C07193=1038.016,139.466,-96.925,169.847,40.558,157.645
C07194=1038.010,139.217,-96.903,169.845,40.559,157.645
C07195=1038.004,138.968,-96.882,169.843,40.558,157.644
C07196=1037.998,138.720,-96.861,169.840,40.559,157.644
C07197=1037.992,138.470,-96.839,169.837,40.558,157.644
C07198=1037.986,138.221,-96.819,169.835,40.558,157.644
C07199=1037.979,137.972,-96.797,169.833,40.558,157.644
C07200=1037.974,137.723,-96.776,169.831,40.558,157.644
C07201=1037.968,137.474,-96.754,169.828,40.558,157.644
C07202=1037.961,137.225,-96.733,169.826,40.557,157.644
C07203=1037.955,136.976,-96.711,169.824,40.558,157.644
C07204=1037.949,136.727,-96.691,169.822,40.557,157.643
C07205=1037.942,136.478,-96.670,169.819,40.557,157.643
C07206=1037.936,136.229,-96.648,169.817,40.557,157.643
C07207=1037.931,135.980,-96.627,169.814,40.557,157.643
C07208=1037.924,135.731,-96.606,169.812,40.557,157.643
C07209=1037.918,135.481,-96.585,169.810,40.557,157.643
C07210=1037.912,135.233,-96.564,169.807,40.557,157.643
C07211=1037.905,134.984,-96.543,169.805,40.556,157.642
C07212=1037.899,134.735,-96.521,169.803,40.557,157.642
C07213=1037.894,134.486,-96.500,169.801,40.556,157.642
C07214=1037.887,134.237,-96.479,169.799,40.556,157.642
C07215=1037.881,133.987,-96.458,169.796,40.556,157.642
C07216=1037.875,133.739,-96.436,169.793,40.556,157.642
C07217=1037.869,133.489,-96.416,169.791,40.556,157.642
C07218=1037.863,133.240,-96.394,169.789,40.555,157.641
C07219=1037.857,132.992,-96.373,169.787,40.556,157.641
C07220=1037.851,132.742,-96.353,169.784,40.555,157.641
C07221=1037.844,132.493,-96.331,169.782,40.556,157.641
C07222=1037.839,132.245,-96.310,169.780,40.555,157.641
C07223=1037.832,131.995,-96.290,169.778,40.555,157.641
C07224=1037.826,131.746,-96.268,169.776,40.555,157.641
C07225=1037.820,131.498,-96.247,169.773,40.555,157.641
C07226=1037.814,131.248,-96.226,169.770,40.555,157.640
C07227=1037.808,130.999,-96.205,169.768,40.554,157.640
C07228=1037.802,130.750,-96.185,169.766,40.555,157.640
C07229=1037.796,130.501,-96.163,169.764,40.554,157.640
C07230=1037.790,130.252,-96.143,169.762,40.554,157.640
C07231=1037.783,130.003,-96.122,169.759,40.555,157.640
C07232=1037.777,129.753,-96.101,169.757,40.554,157.640
C07233=1037.771,129.505,-96.081,169.755,40.555,157.640
C07234=1037.764,129.255,-96.060,169.753,40.554,157.640
C07235=1037.758,129.006,-96.039,169.750,40.554,157.639
C07236=1037.752,128.757,-96.019,169.748,40.555,157.639
C07237=1037.745,128.508,-95.998,169.745,40.554,157.639
C07238=1037.740,128.259,-95.977,169.743,40.554,157.639
C07239=1037.733,128.010,-95.956,169.741,40.554,157.639
C07240=1037.726,127.761,-95.936,169.738,40.554,157.639
C07241=1037.721,127.512,-95.914,169.736,40.555,157.639
C07242=1037.714,127.263,-95.894,169.734,40.554,157.639
C07243=1037.708,127.015,-95.873,169.732,40.554,157.639
C07244=1037.701,126.765,-95.853,169.730,40.554,157.638
C07245=1037.695,126.515,-95.832,169.728,40.554,157.638
C07246=1037.689,126.267,-95.812,169.725,40.554,157.638
C07247=1037.682,126.018,-95.791,169.722,40.554,157.638
C07248=1037.677,125.769,-95.770,169.720,40.554,157.638
C07249=1037.670,125.520,-95.750,169.718,40.554,157.638
C07250=1037.663,125.234,-95.726,169.715,40.554,157.638
C07251=1037.656,124.949,-95.702,169.713,40.554,157.638
C07252=1037.649,124.662,-95.679,169.710,40.554,157.638
C07253=1037.642,124.377,-95.655,169.708,40.554,157.637
C07254=1037.635,124.127,-95.635,169.706,40.554,157.637
C07255=1037.630,123.879,-95.614,169.704,40.554,157.637
C07256=1037.623,123.629,-95.593,169.701,40.554,157.637
C07257=1037.617,123.380,-95.573,169.699,40.554,157.637
C07258=1037.611,123.131,-95.552,169.696,40.554,157.637
C07259=1037.605,122.882,-95.532,169.694,40.554,157.637
C07260=1037.598,122.633,-95.512,169.692,40.554,157.637
C07261=1037.592,122.385,-95.491,169.690,40.554,157.637
C07262=1037.586,122.135,-95.470,169.687,40.554,157.636
C07263=1037.580,121.886,-95.450,169.685,40.553,157.636
C07264=1037.574,121.636,-95.430,169.683,40.554,157.636
C07265=1037.568,121.388,-95.408,169.681,40.553,157.636
C07266=1037.561,121.138,-95.388,169.679,40.553,157.636
C07267=1037.555,120.890,-95.368,169.677,40.554,157.636
C07268=1037.550,120.641,-95.348,169.675,40.553,157.636
C07269=1037.544,120.391,-95.327,169.672,40.554,157.636
C07270=1037.537,120.143,-95.307,169.669,40.553,157.635
C07271=1037.531,119.893,-95.286,169.667,40.553,157.635
C07272=1037.525,119.644,-95.266,169.665,40.553,157.635
C07273=1037.519,119.395,-95.245,169.663,40.553,157.635
C07274=1037.513,119.146,-95.225,169.661,40.553,157.635
C07275=1037.506,118.897,-95.204,169.659,40.553,157.635
C07276=1037.501,118.648,-95.184,169.657,40.553,157.635
C07277=1037.495,118.399,-95.164,169.654,40.553,157.635
C07278=1037.488,118.149,-95.144,169.652,40.553,157.635
C07279=1037.483,117.900,-95.123,169.650,40.553,157.634
C07280=1037.476,117.651,-95.103,169.648,40.553,157.634
C07281=1037.470,117.403,-95.082,169.645,40.552,157.634
C07282=1037.464,117.154,-95.062,169.643,40.553,157.634
C07283=1037.458,116.904,-95.041,169.641,40.552,157.634
C07284=1037.452,116.655,-95.021,169.639,40.552,157.634
C07285=1037.446,116.406,-95.001,169.637,40.553,157.634
C07286=1037.440,116.157,-94.981,169.634,40.552,157.634
C07287=1037.434,115.908,-94.960,169.632,40.552,157.634
C07288=1037.428,115.658,-94.940,169.630,40.552,157.633
C07289=1037.422,115.409,-94.920,169.628,40.552,157.633
C07290=1037.416,115.161,-94.900,169.626,40.552,157.633
C07291=1037.410,114.911,-94.879,169.624,40.552,157.633
C07292=1037.404,114.662,-94.859,169.621,40.552,157.633
C07293=1037.398,114.413,-94.839,169.619,40.552,157.633
C07294=1037.391,114.164,-94.819,169.617,40.551,157.633
C07295=1037.386,113.915,-94.798,169.615,40.552,157.633
C07296=1037.380,113.666,-94.778,169.612,40.551,157.632
C07297=1037.373,113.417,-94.757,169.610,40.551,157.632
C07298=1037.367,113.167,-94.738,169.608,40.552,157.632
C07299=1037.361,112.919,-94.718,169.606,40.551,157.632
C07300=1037.355,112.669,-94.698,169.604,40.551,157.632
C07301=1037.349,112.420,-94.678,169.602,40.552,157.632
C07302=1037.343,112.171,-94.658,169.600,40.551,157.632
C07303=1037.336,111.922,-94.638,169.598,40.551,157.632
C07304=1037.330,111.673,-94.618,169.595,40.552,157.632
C07305=1037.324,111.424,-94.597,169.592,40.551,157.632
C07306=1037.318,111.175,-94.577,169.590,40.552,157.632
C07307=1037.312,110.925,-94.558,169.588,40.552,157.631
C07308=1037.305,110.676,-94.538,169.586,40.551,157.631
C07309=1037.299,110.427,-94.518,169.584,40.552,157.631
C07310=1037.293,110.178,-94.498,169.582,40.552,157.631
C07311=1037.287,109.929,-94.478,169.580,40.551,157.631
C07312=1037.281,109.680,-94.458,169.578,40.552,157.631
C07313=1037.274,109.431,-94.439,169.575,40.552,157.631
C07314=1037.265,109.034,-94.407,169.572,40.552,157.631
C07315=1037.255,108.637,-94.375,169.569,40.552,157.631
C07316=1037.244,108.240,-94.344,169.565,40.552,157.631
C07317=1037.234,107.844,-94.312,169.561,40.552,157.630
C07318=1037.228,107.595,-94.292,169.559,40.552,157.630
C07319=1037.222,107.346,-94.273,169.557,40.552,157.630
C07320=1037.216,107.097,-94.254,169.555,40.552,157.630
C07321=1037.209,106.847,-94.233,169.553,40.552,157.630
C07322=1037.203,106.599,-94.213,169.550,40.553,157.630
C07323=1037.198,106.349,-94.194,169.548,40.552,157.630
C07324=1037.191,106.100,-94.174,169.546,40.552,157.630
C07325=1037.184,105.851,-94.154,169.544,40.553,157.630
C07326=1037.179,105.602,-94.135,169.542,40.553,157.630
C07327=1037.173,105.353,-94.115,169.540,40.552,157.629
C07328=1037.166,105.103,-94.095,169.538,40.553,157.629
C07329=1037.160,104.854,-94.076,169.536,40.553,157.629
C07330=1037.154,104.605,-94.056,169.533,40.552,157.629
C07331=1037.148,104.357,-94.036,169.531,40.553,157.629
C07332=1037.141,104.106,-94.017,169.528,40.553,157.629
C07333=1037.135,103.858,-93.997,169.526,40.552,157.629
C07334=1037.130,103.608,-93.978,169.524,40.553,157.629
C07335=1037.123,103.360,-93.958,169.522,40.553,157.629
C07336=1037.117,103.111,-93.938,169.520,40.553,157.629
C07337=1037.111,102.861,-93.919,169.518,40.553,157.628
C07338=1037.105,102.612,-93.899,169.516,40.553,157.628
C07339=1037.098,102.363,-93.880,169.514,40.553,157.628
C07340=1037.092,102.114,-93.860,169.512,40.553,157.628
C07341=1037.087,101.865,-93.841,169.510,40.553,157.628
C07342=1037.080,101.615,-93.820,169.508,40.553,157.628
C07343=1037.074,101.366,-93.801,169.506,40.553,157.628
C07344=1037.068,101.117,-93.782,169.503,40.553,157.628
C07345=1037.062,100.868,-93.762,169.500,40.553,157.628
C07346=1037.056,100.619,-93.743,169.498,40.553,157.628
C07347=1037.049,100.369,-93.722,169.496,40.553,157.627
C07348=1037.043,100.120,-93.704,169.494,40.553,157.627
C07349=1037.037,99.871,-93.684,169.492,40.553,157.627
C07350=1037.031,99.622,-93.665,169.490,40.553,157.627
C07351=1037.025,99.373,-93.646,169.488,40.553,157.627
C07352=1037.018,99.123,-93.626,169.486,40.553,157.627
C07353=1037.012,98.874,-93.607,169.484,40.554,157.627
C07354=1037.003,98.487,-93.577,169.480,40.554,157.627
C07355=1036.992,98.100,-93.547,169.477,40.554,157.627
C07356=1036.983,97.712,-93.517,169.474,40.554,157.627
C07357=1036.973,97.324,-93.487,169.471,40.554,157.627
C07358=1036.967,97.075,-93.467,169.468,40.554,157.626
C07359=1036.960,96.826,-93.448,169.466,40.554,157.626
C07360=1036.955,96.576,-93.429,169.463,40.554,157.626
C07361=1036.948,96.328,-93.410,169.461,40.555,157.626
C07362=1036.942,96.078,-93.390,169.459,40.555,157.626
C07363=1036.936,95.829,-93.372,169.457,40.554,157.626
C07364=1036.929,95.579,-93.352,169.455,40.555,157.626
C07365=1036.923,95.331,-93.333,169.453,40.555,157.626
C07366=1036.917,95.081,-93.314,169.451,40.555,157.626
C07367=1036.911,94.832,-93.295,169.449,40.555,157.626
C07368=1036.905,94.583,-93.275,169.447,40.555,157.626
C07369=1036.898,94.334,-93.256,169.445,40.555,157.626
C07370=1036.893,94.085,-93.237,169.442,40.555,157.625
C07371=1036.886,93.836,-93.218,169.440,40.556,157.625
C07372=1036.880,93.587,-93.198,169.438,40.555,157.625
C07373=1036.874,93.338,-93.180,169.436,40.555,157.625
C07374=1036.867,93.051,-93.158,169.434,40.556,157.625
C07375=1036.859,92.766,-93.136,169.431,40.556,157.625
C07376=1036.852,92.479,-93.114,169.429,40.555,157.625
C07377=1036.845,92.194,-93.092,169.426,40.556,157.625
C07378=1036.839,91.944,-93.073,169.424,40.556,157.625
C07379=1036.832,91.695,-93.054,169.422,40.556,157.625
C07380=1036.827,91.446,-93.035,169.419,40.556,157.624
C07381=1036.820,91.197,-93.015,169.417,40.556,157.624
C07382=1036.814,90.948,-92.996,169.415,40.556,157.624
C07383=1036.808,90.699,-92.977,169.413,40.556,157.624
C07384=1036.802,90.449,-92.958,169.411,40.556,157.624
C07385=1036.796,90.200,-92.940,169.409,40.556,157.624
C07386=1036.790,89.951,-92.920,169.407,40.556,157.624
C07387=1036.784,89.702,-92.902,169.405,40.557,157.624
C07388=1036.777,89.452,-92.883,169.403,40.557,157.624
C07389=1036.771,89.203,-92.864,169.401,40.556,157.624
C07390=1036.765,88.954,-92.844,169.399,40.557,157.624
C07391=1036.758,88.705,-92.826,169.397,40.557,157.624
C07392=1036.752,88.456,-92.807,169.395,40.557,157.624
C07393=1036.746,88.207,-92.788,169.392,40.557,157.623
C07394=1036.739,87.958,-92.770,169.390,40.558,157.623
C07395=1036.733,87.708,-92.750,169.388,40.558,157.623
C07396=1036.726,87.459,-92.732,169.386,40.558,157.623
C07397=1036.720,87.210,-92.713,169.384,40.558,157.623
C07398=1036.714,86.960,-92.694,169.381,40.558,157.623
C07399=1036.707,86.711,-92.676,169.379,40.558,157.623
C07400=1036.701,86.462,-92.656,169.377,40.558,157.623
C07401=1036.695,86.213,-92.638,169.375,40.558,157.623
C07402=1036.689,85.963,-92.620,169.373,40.559,157.623
C07403=1036.682,85.714,-92.601,169.371,40.559,157.623
C07404=1036.676,85.465,-92.582,169.368,40.559,157.623
C07405=1036.670,85.215,-92.563,169.366,40.559,157.623
C07406=1036.664,84.966,-92.545,169.364,40.559,157.623
C07407=1036.657,84.717,-92.526,169.362,40.559,157.622
C07408=1036.651,84.468,-92.507,169.360,40.559,157.622
C07409=1036.645,84.219,-92.489,169.358,40.560,157.622
C07410=1036.638,83.970,-92.470,169.356,40.560,157.622
C07411=1036.633,83.720,-92.451,169.354,40.560,157.622
C07412=1036.626,83.471,-92.432,169.352,40.560,157.622
C07413=1036.620,83.221,-92.414,169.350,40.560,157.622
C07414=1036.614,82.973,-92.396,169.348,40.560,157.622
C07415=1036.608,82.724,-92.377,169.346,40.560,157.622
C07416=1036.602,82.475,-92.358,169.344,40.560,157.622
C07417=1036.596,82.225,-92.339,169.341,40.561,157.622
C07418=1036.589,81.976,-92.321,169.338,40.560,157.622
C07419=1036.583,81.727,-92.302,169.336,40.561,157.622
C07420=1036.577,81.477,-92.284,169.334,40.561,157.621
C07421=1036.570,81.228,-92.265,169.332,40.561,157.621
C07422=1036.565,80.979,-92.246,169.330,40.561,157.621
C07423=1036.558,80.730,-92.228,169.328,40.561,157.621
C07424=1036.552,80.481,-92.209,169.326,40.561,157.621
C07425=1036.546,80.231,-92.191,169.324,40.561,157.621
C07426=1036.539,79.982,-92.172,169.322,40.561,157.621
C07427=1036.533,79.733,-92.154,169.320,40.562,157.621
C07428=1036.528,79.484,-92.135,169.318,40.562,157.621
C07429=1036.521,79.235,-92.116,169.316,40.561,157.621
C07430=1036.515,78.985,-92.098,169.314,40.562,157.621
C07431=1036.509,78.736,-92.080,169.312,40.562,157.621
C07432=1036.502,78.487,-92.061,169.310,40.562,157.621
C07433=1036.496,78.237,-92.043,169.307,40.562,157.621
C07434=1036.490,77.988,-92.024,169.305,40.563,157.620
C07435=1036.483,77.739,-92.006,169.303,40.562,157.620
C07436=1036.477,77.490,-91.987,169.301,40.562,157.620
C07437=1036.471,77.241,-91.969,169.299,40.563,157.620
C07438=1036.464,76.954,-91.948,169.297,40.563,157.620
C07439=1036.457,76.669,-91.927,169.293,40.563,157.620
C07440=1036.450,76.383,-91.906,169.291,40.563,157.620
C07441=1036.442,76.096,-91.885,169.289,40.564,157.620
C07442=1036.436,75.848,-91.867,169.287,40.564,157.620
C07443=1036.430,75.599,-91.848,169.284,40.564,157.620
C07444=1036.424,75.349,-91.830,169.282,40.564,157.620
C07445=1036.417,75.100,-91.812,169.280,40.564,157.620
C07446=1036.411,74.850,-91.794,169.278,40.564,157.620
C07447=1036.405,74.601,-91.775,169.276,40.564,157.619
C07448=1036.398,74.351,-91.758,169.274,40.564,157.619
C07449=1036.392,74.103,-91.740,169.272,40.565,157.619
C07450=1036.386,73.854,-91.721,169.270,40.565,157.619
C07451=1036.380,73.604,-91.703,169.268,40.565,157.619
C07452=1036.373,73.355,-91.684,169.266,40.565,157.619
C07453=1036.367,73.105,-91.666,169.264,40.566,157.619
C07454=1036.361,72.856,-91.648,169.262,40.566,157.619
C07455=1036.355,72.607,-91.630,169.259,40.566,157.619
C07456=1036.348,72.358,-91.612,169.257,40.566,157.619
C07457=1036.342,72.108,-91.594,169.255,40.566,157.619
C07458=1036.335,71.859,-91.576,169.253,40.566,157.619
C07459=1036.329,71.610,-91.558,169.251,40.566,157.619
C07460=1036.323,71.361,-91.539,169.249,40.566,157.619
C07461=1036.317,71.111,-91.521,169.247,40.567,157.619
C07462=1036.311,70.862,-91.503,169.245,40.567,157.619
C07463=1036.304,70.613,-91.485,169.243,40.567,157.618
C07464=1036.298,70.363,-91.467,169.241,40.567,157.618
C07465=1036.292,70.115,-91.449,169.239,40.568,157.618
C07466=1036.286,69.865,-91.431,169.237,40.568,157.618
C07467=1036.280,69.616,-91.413,169.234,40.567,157.618
C07468=1036.273,69.366,-91.395,169.231,40.568,157.618
C07469=1036.267,69.117,-91.378,169.229,40.568,157.618
C07470=1036.261,68.868,-91.359,169.227,40.568,157.618
C07471=1036.255,68.619,-91.341,169.225,40.568,157.618
C07472=1036.249,68.369,-91.323,169.223,40.568,157.618
C07473=1036.241,68.120,-91.305,169.221,40.569,157.618
C07474=1036.236,67.871,-91.288,169.219,40.569,157.618
C07475=1036.230,67.621,-91.270,169.217,40.569,157.618
C07476=1036.223,67.372,-91.252,169.215,40.569,157.618
C07477=1036.216,67.123,-91.234,169.213,40.570,157.618
C07478=1036.211,66.874,-91.216,169.211,40.570,157.617
C07479=1036.204,66.625,-91.197,169.209,40.570,157.617
C07480=1036.198,66.375,-91.180,169.206,40.570,157.617
C07481=1036.192,66.125,-91.162,169.204,40.571,157.617
C07482=1036.186,65.877,-91.144,169.202,40.571,157.617
C07483=1036.179,65.627,-91.127,169.200,40.571,157.617
C07484=1036.173,65.378,-91.109,169.198,40.570,157.617
C07485=1036.166,65.129,-91.092,169.196,40.571,157.617
C07486=1036.160,64.880,-91.073,169.194,40.571,157.617
C07487=1036.154,64.630,-91.055,169.192,40.571,157.617
C07488=1036.147,64.381,-91.038,169.190,40.571,157.617
C07489=1036.142,64.132,-91.020,169.188,40.572,157.617
C07490=1036.135,63.882,-91.002,169.186,40.572,157.617
C07491=1036.128,63.633,-90.984,169.183,40.572,157.617
C07492=1036.122,63.383,-90.966,169.181,40.572,157.617
C07493=1036.116,63.135,-90.949,169.179,40.573,157.617
C07494=1036.109,62.885,-90.932,169.177,40.573,157.616
C07495=1036.103,62.635,-90.914,169.175,40.574,157.617
C07496=1036.097,62.387,-90.897,169.173,40.574,157.616
C07497=1036.091,62.137,-90.879,169.171,40.574,157.616
C07498=1036.084,61.888,-90.862,169.169,40.574,157.616
C07499=1036.077,61.638,-90.844,169.166,40.575,157.616
C07500=1036.071,61.389,-90.827,169.164,40.575,157.616
C07501=1036.064,61.140,-90.809,169.162,40.575,157.616
C07502=1036.057,60.854,-90.789,169.160,40.575,157.616
C07503=1036.050,60.568,-90.768,169.156,40.576,157.616
C07504=1036.043,60.282,-90.749,169.154,40.576,157.616
C07505=1036.034,59.995,-90.729,169.151,40.576,157.616
C07506=1036.029,59.746,-90.711,169.150,40.577,157.616
C07507=1036.022,59.497,-90.694,169.148,40.577,157.616
C07508=1036.015,59.248,-90.677,169.146,40.577,157.616
C07509=1036.010,58.999,-90.659,169.143,40.578,157.616
C07510=1036.003,58.749,-90.642,169.141,40.578,157.616
C07511=1035.997,58.499,-90.624,169.139,40.578,157.616
C07512=1035.990,58.251,-90.607,169.136,40.578,157.616
C07513=1035.983,58.001,-90.589,169.134,40.579,157.616
C07514=1035.977,57.751,-90.571,169.132,40.579,157.616
C07515=1035.971,57.503,-90.555,169.130,40.579,157.615
C07516=1035.964,57.253,-90.537,169.128,40.579,157.615
C07517=1035.958,57.003,-90.520,169.126,40.579,157.615
C07518=1035.952,56.754,-90.503,169.124,40.580,157.615
C07519=1035.945,56.505,-90.486,169.122,40.580,157.615
C07520=1035.939,56.255,-90.468,169.120,40.580,157.615
C07521=1035.933,56.006,-90.451,169.117,40.580,157.615
C07522=1035.926,55.757,-90.433,169.115,40.581,157.615
C07523=1035.921,55.508,-90.416,169.113,40.581,157.615
C07524=1035.914,55.258,-90.399,169.111,40.581,157.615
C07525=1035.907,55.009,-90.381,169.109,40.581,157.615
C07526=1035.901,54.760,-90.364,169.107,40.582,157.615
C07527=1035.895,54.510,-90.347,169.105,40.582,157.615
C07528=1035.889,54.261,-90.330,169.103,40.582,157.615
C07529=1035.882,54.011,-90.312,169.100,40.583,157.615
C07530=1035.876,53.763,-90.295,169.098,40.583,157.615
C07531=1035.869,53.513,-90.278,169.096,40.583,157.615
C07532=1035.863,53.264,-90.260,169.094,40.583,157.615
C07533=1035.857,53.015,-90.243,169.092,40.584,157.615
C07534=1035.850,52.765,-90.226,169.090,40.584,157.615
C07535=1035.845,52.516,-90.209,169.088,40.584,157.614
C07536=1035.838,52.266,-90.191,169.086,40.584,157.614
C07537=1035.832,52.018,-90.174,169.084,40.584,157.614
C07538=1035.826,51.768,-90.156,169.081,40.585,157.614
C07539=1035.820,51.518,-90.140,169.079,40.585,157.614
C07540=1035.813,51.269,-90.123,169.077,40.585,157.614
C07541=1035.807,51.020,-90.105,169.075,40.585,157.614
C07542=1035.800,50.771,-90.088,169.073,40.586,157.614
C07543=1035.794,50.521,-90.072,169.071,40.586,157.614
C07544=1035.788,50.272,-90.054,169.069,40.586,157.614
C07545=1035.782,50.023,-90.037,169.067,40.586,157.614
C07546=1035.775,49.773,-90.019,169.065,40.587,157.614
C07547=1035.769,49.524,-90.003,169.063,40.587,157.614
C07548=1035.763,49.274,-89.985,169.060,40.586,157.614
C07549=1035.757,49.025,-89.968,169.058,40.587,157.614
C07550=1035.750,48.776,-89.951,169.055,40.587,157.613
C07551=1035.745,48.526,-89.934,169.053,40.587,157.613
C07552=1035.738,48.277,-89.917,169.051,40.587,157.613
C07553=1035.732,48.028,-89.900,169.049,40.587,157.613
C07554=1035.725,47.778,-89.883,169.047,40.588,157.613
C07555=1035.720,47.529,-89.866,169.045,40.588,157.613
C07556=1035.713,47.280,-89.849,169.043,40.588,157.613
C07557=1035.707,47.030,-89.832,169.040,40.588,157.613
C07558=1035.701,46.781,-89.814,169.038,40.589,157.613
C07559=1035.694,46.532,-89.797,169.036,40.589,157.613
C07560=1035.688,46.283,-89.781,169.034,40.589,157.613
C07561=1035.682,46.033,-89.763,169.032,40.589,157.613
C07562=1035.676,45.784,-89.746,169.030,40.589,157.613
C07563=1035.670,45.535,-89.730,169.028,40.590,157.613
C07564=1035.663,45.285,-89.712,169.026,40.590,157.613
C07565=1035.658,45.036,-89.695,169.024,40.590,157.613
C07566=1035.650,44.749,-89.676,169.021,40.590,157.613
C07567=1035.643,44.463,-89.657,169.019,40.591,157.613
C07568=1035.636,44.177,-89.637,169.016,40.590,157.612
C07569=1035.630,43.890,-89.617,169.014,40.591,157.612
C07570=1035.623,43.640,-89.601,169.012,40.591,157.612
C07571=1035.617,43.391,-89.584,169.010,40.591,157.612
C07572=1035.611,43.142,-89.566,169.008,40.591,157.612
C07573=1035.605,42.892,-89.550,169.006,40.591,157.612
C07574=1035.599,42.643,-89.533,169.003,40.592,157.612
C07575=1035.592,42.394,-89.516,169.001,40.592,157.612
C07576=1035.586,42.144,-89.500,168.999,40.592,157.612
C07577=1035.579,41.895,-89.482,168.997,40.592,157.612
C07578=1035.573,41.645,-89.466,168.995,40.593,157.612
C07579=1035.567,41.397,-89.449,168.993,40.593,157.612
C07580=1035.560,41.147,-89.432,168.991,40.594,157.612
C07581=1035.554,40.898,-89.416,168.988,40.594,157.612
C07582=1035.547,40.648,-89.399,168.986,40.594,157.612
C07583=1035.541,40.399,-89.383,168.984,40.594,157.612
C07584=1035.535,40.150,-89.366,168.982,40.595,157.612
C07585=1035.529,39.900,-89.349,168.980,40.595,157.611
C07586=1035.522,39.651,-89.332,168.978,40.595,157.611
C07587=1035.516,39.402,-89.316,168.976,40.595,157.611
C07588=1035.510,39.152,-89.299,168.973,40.596,157.611
C07589=1035.504,38.903,-89.282,168.970,40.596,157.611
C07590=1035.498,38.654,-89.266,168.968,40.596,157.611
C07591=1035.491,38.404,-89.249,168.966,40.596,157.611
C07592=1035.485,38.155,-89.232,168.964,40.596,157.611
C07593=1035.479,37.905,-89.216,168.962,40.597,157.611
C07594=1035.472,37.655,-89.199,168.960,40.597,157.611
C07595=1035.466,37.407,-89.183,168.957,40.597,157.611
C07596=1035.460,37.157,-89.166,168.955,40.597,157.611
C07597=1035.454,36.907,-89.150,168.953,40.598,157.611
C07598=1035.447,36.658,-89.134,168.951,40.598,157.611
C07599=1035.441,36.410,-89.117,168.949,40.599,157.611
C07600=1035.434,36.159,-89.100,168.947,40.599,157.611
C07601=1035.428,35.910,-89.084,168.944,40.599,157.611
C07602=1035.422,35.661,-89.068,168.942,40.599,157.611
C07603=1035.415,35.411,-89.052,168.940,40.600,157.611
C07604=1035.409,35.162,-89.035,168.938,40.600,157.611
C07605=1035.403,34.913,-89.019,168.936,40.601,157.611
C07606=1035.396,34.663,-89.002,168.934,40.601,157.610
C07607=1035.390,34.414,-88.986,168.931,40.601,157.610
C07608=1035.384,34.165,-88.970,168.929,40.601,157.610
C07609=1035.377,33.915,-88.953,168.927,40.602,157.610
C07610=1035.371,33.666,-88.936,168.925,40.602,157.610
C07611=1035.365,33.416,-88.920,168.923,40.603,157.610
C07612=1035.358,33.167,-88.905,168.920,40.603,157.610
C07613=1035.352,32.917,-88.888,168.918,40.603,157.610
C07614=1035.346,32.668,-88.872,168.916,40.603,157.610
C07615=1035.340,32.419,-88.855,168.914,40.604,157.610
C07616=1035.333,32.170,-88.840,168.912,40.604,157.610
C07617=1035.326,31.920,-88.822,168.910,40.604,157.610
C07618=1035.320,31.671,-88.806,168.907,40.604,157.610
C07619=1035.314,31.421,-88.790,168.905,40.605,157.610
C07620=1035.308,31.172,-88.774,168.903,40.605,157.610
C07621=1035.301,30.922,-88.758,168.901,40.606,157.610
C07622=1035.295,30.673,-88.741,168.899,40.606,157.610
C07623=1035.289,30.424,-88.725,168.896,40.606,157.610
C07624=1035.282,30.175,-88.709,168.894,40.606,157.610
C07625=1035.276,29.925,-88.693,168.892,40.607,157.610
C07626=1035.270,29.675,-88.677,168.890,40.607,157.610
C07627=1035.264,29.426,-88.660,168.888,40.607,157.609
C07628=1035.257,29.177,-88.645,168.886,40.607,157.609
C07629=1035.251,28.927,-88.628,168.883,40.608,157.609
C07630=1035.244,28.641,-88.610,168.881,40.608,157.609
C07631=1035.237,28.354,-88.590,168.878,40.609,157.609
C07632=1035.230,28.067,-88.572,168.876,40.609,157.609
C07633=1035.222,27.781,-88.554,168.873,40.609,157.609
C07634=1035.215,27.532,-88.538,168.871,40.610,157.609
C07635=1035.209,27.282,-88.522,168.869,40.610,157.609
C07636=1035.203,27.033,-88.506,168.867,40.611,157.609
C07637=1035.197,26.784,-88.490,168.865,40.611,157.609
C07638=1035.190,26.534,-88.473,168.862,40.611,157.609
C07639=1035.184,26.284,-88.458,168.860,40.611,157.609
C07640=1035.178,26.035,-88.442,168.858,40.612,157.609
C07641=1035.171,25.786,-88.426,168.856,40.612,157.609
C07642=1035.165,25.537,-88.410,168.853,40.613,157.609
C07643=1035.158,25.287,-88.394,168.851,40.613,157.609
C07644=1035.152,25.038,-88.378,168.849,40.613,157.609
C07645=1035.145,24.789,-88.362,168.847,40.613,157.609
C07646=1035.140,24.539,-88.347,168.845,40.614,157.609
C07647=1035.133,24.290,-88.331,168.842,40.615,157.609
C07648=1035.127,24.040,-88.315,168.840,40.615,157.609
C07649=1035.120,23.791,-88.299,168.838,40.615,157.609
C07650=1035.114,23.541,-88.282,168.836,40.615,157.609
C07651=1035.107,23.292,-88.267,168.833,40.616,157.608
C07652=1035.102,23.042,-88.251,168.831,40.616,157.609
C07653=1035.095,22.793,-88.235,168.829,40.617,157.608
C07654=1035.089,22.544,-88.219,168.827,40.617,157.608
C07655=1035.082,22.295,-88.204,168.825,40.617,157.608
C07656=1035.077,22.045,-88.188,168.822,40.617,157.608
C07657=1035.070,21.796,-88.172,168.820,40.618,157.608
C07658=1035.063,21.546,-88.156,168.818,40.618,157.608
C07659=1035.057,21.297,-88.140,168.816,40.619,157.608
C07660=1035.051,21.047,-88.125,168.813,40.619,157.608
C07661=1035.044,20.798,-88.109,168.811,40.619,157.608
C07662=1035.038,20.548,-88.093,168.809,40.619,157.608
C07663=1035.032,20.299,-88.077,168.807,40.620,157.608
C07664=1035.026,20.049,-88.061,168.805,40.621,157.608
C07665=1035.019,19.800,-88.046,168.802,40.621,157.608
C07666=1035.013,19.551,-88.029,168.800,40.621,157.608
C07667=1035.007,19.301,-88.015,168.798,40.621,157.608
C07668=1035.000,19.052,-87.999,168.796,40.621,157.608
C07669=1034.995,18.802,-87.983,168.793,40.622,157.608
C07670=1034.987,18.552,-87.967,168.791,40.623,157.608
C07671=1034.981,18.303,-87.952,168.789,40.623,157.608
C07672=1034.975,18.053,-87.936,168.787,40.623,157.608
C07673=1034.968,17.804,-87.920,168.784,40.624,157.608
C07674=1034.962,17.555,-87.905,168.782,40.624,157.608
C07675=1034.956,17.305,-87.889,168.780,40.625,157.608
C07676=1034.949,17.056,-87.874,168.778,40.625,157.608
C07677=1034.944,16.806,-87.858,168.775,40.625,157.607
C07678=1034.937,16.557,-87.842,168.773,40.626,157.608
C07679=1034.931,16.308,-87.827,168.771,40.626,157.608
C07680=1034.925,16.058,-87.811,168.769,40.626,157.607
C07681=1034.918,15.809,-87.796,168.766,40.627,157.607
C07682=1034.912,15.560,-87.781,168.764,40.627,157.607
C07683=1034.906,15.310,-87.764,168.762,40.628,157.607
C07684=1034.899,15.061,-87.749,168.760,40.628,157.607
C07685=1034.893,14.812,-87.734,168.757,40.628,157.607
C07686=1034.887,14.562,-87.718,168.755,40.628,157.607
C07687=1034.880,14.313,-87.702,168.753,40.629,157.607
C07688=1034.874,14.063,-87.688,168.751,40.630,157.607
C07689=1034.868,13.813,-87.672,168.748,40.630,157.607
C07690=1034.862,13.564,-87.656,168.746,40.630,157.607
C07691=1034.855,13.314,-87.641,168.744,40.631,157.607
C07692=1034.848,13.065,-87.626,168.741,40.631,157.607
C07693=1034.842,12.816,-87.611,168.739,40.632,157.607
C07694=1034.835,12.530,-87.593,168.737,40.632,157.607
C07695=1034.827,12.245,-87.575,168.734,40.633,157.607
C07696=1034.820,11.959,-87.558,168.731,40.633,157.607
C07697=1034.813,11.675,-87.541,168.729,40.634,157.607
C07698=1034.806,11.425,-87.526,168.726,40.634,157.607
C07699=1034.800,11.176,-87.511,168.725,40.635,157.607
C07700=1034.793,10.926,-87.496,168.723,40.635,157.607
C07701=1034.787,10.677,-87.481,168.719,40.636,157.607
C07702=1034.780,10.428,-87.465,168.718,40.636,157.607
C07703=1034.774,10.178,-87.450,168.716,40.637,157.607
C07704=1034.768,9.928,-87.435,168.713,40.637,157.607
C07705=1034.761,9.679,-87.419,168.711,40.638,157.607
C07706=1034.754,9.430,-87.404,168.709,40.638,157.607
C07707=1034.749,9.180,-87.389,168.707,40.638,157.607
C07708=1034.742,8.930,-87.374,168.704,40.639,157.607
C07709=1034.736,8.681,-87.358,168.702,40.640,157.607
C07710=1034.729,8.431,-87.343,168.700,40.640,157.607
C07711=1034.723,8.182,-87.328,168.697,40.640,157.607
C07712=1034.717,7.932,-87.313,168.695,40.641,157.607
C07713=1034.710,7.683,-87.298,168.693,40.641,157.607
C07714=1034.704,7.433,-87.283,168.690,40.641,157.606
C07715=1034.698,7.184,-87.268,168.688,40.642,157.607
C07716=1034.691,6.935,-87.253,168.686,40.643,157.607
C07717=1034.685,6.686,-87.238,168.683,40.643,157.606
C07718=1034.678,6.436,-87.223,168.681,40.644,157.606
C07719=1034.672,6.186,-87.208,168.679,40.644,157.606
C07720=1034.665,5.937,-87.193,168.676,40.644,157.606
C07721=1034.659,5.687,-87.178,168.674,40.644,157.606
C07722=1034.652,5.438,-87.162,168.672,40.645,157.606
C07723=1034.647,5.189,-87.148,168.670,40.646,157.606
C07724=1034.640,4.939,-87.133,168.667,40.646,157.606
C07725=1034.634,4.690,-87.118,168.665,40.647,157.606
C07726=1034.627,4.440,-87.103,168.663,40.647,157.606
C07727=1034.621,4.191,-87.088,168.660,40.647,157.606
C07728=1034.615,3.941,-87.073,168.658,40.648,157.606
C07729=1034.609,3.692,-87.058,168.656,40.648,157.606
C07730=1034.602,3.443,-87.043,168.653,40.649,157.606
C07731=1034.597,3.193,-87.027,168.651,40.649,157.606
C07732=1034.590,2.943,-87.012,168.649,40.650,157.606
C07733=1034.584,2.694,-86.997,168.646,40.650,157.606
C07734=1034.577,2.444,-86.982,168.644,40.650,157.606
C07735=1034.572,2.195,-86.968,168.642,40.651,157.606
C07736=1034.565,1.945,-86.953,168.639,40.652,157.606
C07737=1034.559,1.696,-86.938,168.637,40.652,157.606
C07738=1034.553,1.446,-86.923,168.635,40.652,157.606
C07739=1034.547,1.197,-86.908,168.632,40.653,157.606
C07740=1034.540,0.947,-86.893,168.630,40.653,157.606
C07741=1034.534,0.698,-86.878,168.628,40.653,157.606
C07742=1034.528,0.448,-86.863,168.625,40.654,157.606
C07743=1034.521,0.198,-86.849,168.623,40.655,157.606
C07744=1034.515,-0.051,-86.834,168.621,40.655,157.606
C07745=1034.509,-0.300,-86.819,168.618,40.655,157.606
C07746=1034.503,-0.550,-86.804,168.616,40.655,157.606
C07747=1034.496,-0.800,-86.789,168.614,40.656,157.606
C07748=1034.491,-1.048,-86.775,168.612,40.656,157.606
C07749=1034.484,-1.298,-86.760,168.609,40.657,157.605
C07750=1034.478,-1.548,-86.745,168.607,40.657,157.605
C07751=1034.472,-1.797,-86.730,168.605,40.658,157.605
C07752=1034.466,-2.046,-86.715,168.602,40.658,157.605
C07753=1034.459,-2.296,-86.700,168.600,40.658,157.605
C07754=1034.453,-2.546,-86.685,168.598,40.659,157.605
C07755=1034.447,-2.795,-86.671,168.595,40.660,157.605
C07756=1034.441,-3.044,-86.656,168.593,40.660,157.605
C07757=1034.434,-3.294,-86.641,168.591,40.660,157.605
C07758=1034.427,-3.577,-86.624,168.588,40.660,157.605
C07759=1034.420,-3.861,-86.608,168.585,40.661,157.605
C07760=1034.413,-4.144,-86.592,168.582,40.662,157.605
C07761=1034.406,-4.427,-86.575,168.580,40.662,157.605
C07762=1034.399,-4.677,-86.561,168.577,40.663,157.605
C07763=1034.393,-4.926,-86.546,168.576,40.664,157.605
C07764=1034.387,-5.176,-86.531,168.574,40.664,157.605
C07765=1034.380,-5.425,-86.517,168.571,40.664,157.605
C07766=1034.374,-5.674,-86.503,168.569,40.665,157.605
C07767=1034.368,-5.924,-86.488,168.566,40.665,157.605
C07768=1034.361,-6.174,-86.474,168.564,40.666,157.605
C07769=1034.354,-6.423,-86.459,168.562,40.666,157.605
C07770=1034.349,-6.673,-86.445,168.559,40.667,157.605
C07771=1034.342,-6.922,-86.431,168.557,40.668,157.605
C07772=1034.335,-7.172,-86.416,168.554,40.668,157.605
C07773=1034.329,-7.421,-86.401,168.552,40.669,157.605
C07774=1034.323,-7.671,-86.388,168.550,40.669,157.605
C07775=1034.316,-7.921,-86.373,168.547,40.670,157.605
C07776=1034.310,-8.170,-86.358,168.545,40.670,157.605
C07777=1034.304,-8.419,-86.344,168.542,40.671,157.605
C07778=1034.297,-8.669,-86.330,168.540,40.671,157.605
C07779=1034.291,-8.918,-86.316,168.538,40.672,157.605
C07780=1034.285,-9.168,-86.301,168.535,40.673,157.605
C07781=1034.279,-9.417,-86.287,168.533,40.673,157.605
C07782=1034.272,-9.667,-86.273,168.530,40.674,157.605
C07783=1034.266,-9.917,-86.258,168.528,40.674,157.605
C07784=1034.260,-10.166,-86.244,168.525,40.674,157.605
C07785=1034.253,-10.416,-86.230,168.523,40.675,157.605
C07786=1034.247,-10.665,-86.215,168.521,40.675,157.605
C07787=1034.241,-10.915,-86.201,168.518,40.676,157.605
C07788=1034.234,-11.164,-86.187,168.516,40.677,157.605
C07789=1034.228,-11.413,-86.172,168.513,40.677,157.605
C07790=1034.221,-11.663,-86.159,168.511,40.678,157.605
C07791=1034.216,-11.912,-86.144,168.509,40.678,157.605
C07792=1034.210,-12.162,-86.130,168.507,40.679,157.605
C07793=1034.202,-12.412,-86.115,168.504,40.679,157.605
C07794=1034.197,-12.661,-86.102,168.501,40.680,157.605
C07795=1034.191,-12.911,-86.087,168.500,40.680,157.605
C07796=1034.184,-13.160,-86.073,168.497,40.681,157.605
C07797=1034.178,-13.410,-86.058,168.495,40.682,157.605
C07798=1034.172,-13.659,-86.045,168.493,40.682,157.605
C07799=1034.165,-13.909,-86.030,168.490,40.682,157.604
C07800=1034.160,-14.158,-86.016,168.488,40.683,157.605
C07801=1034.153,-14.408,-86.002,168.485,40.683,157.604
C07802=1034.147,-14.657,-85.988,168.483,40.684,157.604
C07803=1034.140,-14.907,-85.974,168.481,40.684,157.604
C07804=1034.135,-15.156,-85.960,168.478,40.685,157.604
C07805=1034.128,-15.406,-85.945,168.476,40.686,157.604
C07806=1034.122,-15.655,-85.932,168.473,40.686,157.604
C07807=1034.115,-15.905,-85.918,168.471,40.687,157.604
C07808=1034.109,-16.155,-85.903,168.468,40.687,157.604
C07809=1034.103,-16.404,-85.890,168.466,40.688,157.604
C07810=1034.096,-16.654,-85.876,168.463,40.688,157.604
C07811=1034.090,-16.903,-85.862,168.461,40.689,157.604
C07812=1034.083,-17.153,-85.848,168.458,40.690,157.604
C07813=1034.078,-17.402,-85.834,168.456,40.690,157.604
C07814=1034.071,-17.652,-85.820,168.453,40.691,157.604
C07815=1034.065,-17.901,-85.806,168.451,40.692,157.604
C07816=1034.058,-18.151,-85.792,168.448,40.693,157.604
C07817=1034.052,-18.400,-85.778,168.446,40.693,157.604
C07818=1034.045,-18.650,-85.765,168.444,40.694,157.604
C07819=1034.040,-18.899,-85.751,168.441,40.694,157.604
C07820=1034.033,-19.149,-85.736,168.440,40.695,157.604
C07821=1034.026,-19.398,-85.723,168.437,40.695,157.604
C07822=1034.019,-19.681,-85.708,168.434,40.696,157.604
C07823=1034.012,-19.962,-85.692,168.431,40.697,157.604
C07824=1034.005,-20.243,-85.676,168.429,40.697,157.604
C07825=1033.998,-20.525,-85.661,168.426,40.698,157.604
C07826=1033.992,-20.775,-85.647,168.423,40.699,157.604
C07827=1033.985,-21.024,-85.633,168.421,40.700,157.604
C07828=1033.979,-21.273,-85.619,168.418,40.700,157.604
C07829=1033.973,-21.524,-85.605,168.416,40.701,157.604
C07830=1033.967,-21.773,-85.592,168.413,40.701,157.604
C07831=1033.960,-22.023,-85.578,168.411,40.702,157.604
C07832=1033.955,-22.272,-85.564,168.408,40.702,157.604
C07833=1033.948,-22.521,-85.550,168.406,40.703,157.604
C07834=1033.941,-22.771,-85.537,168.403,40.704,157.604
C07835=1033.935,-23.020,-85.523,168.401,40.704,157.604
C07836=1033.929,-23.271,-85.509,168.398,40.705,157.604
C07837=1033.923,-23.520,-85.496,168.396,40.706,157.604
C07838=1033.917,-23.769,-85.483,168.393,40.706,157.604
C07839=1033.911,-24.019,-85.468,168.391,40.707,157.604
C07840=1033.904,-24.268,-85.455,168.388,40.707,157.604
C07841=1033.898,-24.517,-85.441,168.387,40.708,157.604
C07842=1033.892,-24.768,-85.427,168.384,40.708,157.604
C07843=1033.885,-25.017,-85.414,168.382,40.709,157.604
C07844=1033.879,-25.266,-85.400,168.379,40.710,157.604
C07845=1033.873,-25.516,-85.386,168.377,40.710,157.604
C07846=1033.867,-25.766,-85.373,168.374,40.711,157.604
C07847=1033.861,-26.015,-85.360,168.372,40.712,157.604
C07848=1033.855,-26.265,-85.345,168.369,40.712,157.604
C07849=1033.848,-26.514,-85.332,168.367,40.713,157.604
C07850=1033.842,-26.764,-85.319,168.364,40.713,157.604
C07851=1033.835,-27.014,-85.305,168.362,40.714,157.604
C07852=1033.830,-27.263,-85.291,168.359,40.714,157.604
C07853=1033.824,-27.513,-85.278,168.357,40.715,157.604
C07854=1033.817,-27.763,-85.265,168.354,40.716,157.604
C07855=1033.811,-28.012,-85.251,168.352,40.716,157.604
C07856=1033.804,-28.261,-85.238,168.349,40.717,157.604
C07857=1033.798,-28.511,-85.224,168.347,40.718,157.604
C07858=1033.791,-28.760,-85.211,168.344,40.719,157.604
C07859=1033.785,-29.010,-85.198,168.343,40.720,157.604
C07860=1033.779,-29.260,-85.185,168.340,40.721,157.604
C07861=1033.773,-29.509,-85.172,168.337,40.721,157.604
C07862=1033.766,-29.759,-85.158,168.335,40.722,157.604
C07863=1033.760,-30.009,-85.145,168.332,40.722,157.604
C07864=1033.753,-30.258,-85.131,168.330,40.723,157.604
C07865=1033.747,-30.507,-85.118,168.327,40.724,157.604
C07866=1033.741,-30.756,-85.105,168.325,40.724,157.604
C07867=1033.734,-31.007,-85.092,168.322,40.725,157.604
C07868=1033.728,-31.256,-85.079,168.319,40.726,157.604
C07869=1033.722,-31.505,-85.065,168.317,40.726,157.604
C07870=1033.715,-31.755,-85.052,168.314,40.727,157.604
C07871=1033.709,-32.005,-85.039,168.312,40.728,157.604
C07872=1033.704,-32.255,-85.025,168.309,40.729,157.604
C07873=1033.698,-32.504,-85.012,168.307,40.729,157.604
C07874=1033.691,-32.753,-84.999,168.305,40.730,157.604
C07875=1033.684,-33.003,-84.985,168.301,40.731,157.604
C07876=1033.679,-33.253,-84.973,168.300,40.732,157.604
C07877=1033.672,-33.503,-84.959,168.297,40.732,157.604
C07878=1033.666,-33.752,-84.946,168.295,40.733,157.604
C07879=1033.659,-34.002,-84.932,168.292,40.734,157.604
C07880=1033.653,-34.252,-84.920,168.290,40.734,157.604
C07881=1033.647,-34.501,-84.907,168.287,40.735,157.604
C07882=1033.641,-34.750,-84.893,168.284,40.736,157.604
C07883=1033.635,-34.999,-84.880,168.282,40.736,157.604
C07884=1033.629,-35.249,-84.868,168.279,40.737,157.604
C07885=1033.622,-35.499,-84.854,168.277,40.738,157.604
C07886=1033.615,-35.780,-84.840,168.274,40.738,157.604
C07887=1033.608,-36.061,-84.825,168.271,40.739,157.604
C07888=1033.602,-36.342,-84.810,168.268,40.740,157.604
C07889=1033.594,-36.623,-84.796,168.265,40.741,157.604
C07890=1033.588,-36.873,-84.782,168.262,40.742,157.604
C07891=1033.582,-37.122,-84.769,168.261,40.743,157.604
C07892=1033.576,-37.372,-84.757,168.258,40.743,157.604
C07893=1033.570,-37.621,-84.743,168.256,40.744,157.604
C07894=1033.563,-37.871,-84.730,168.253,40.744,157.604
C07895=1033.557,-38.121,-84.717,168.251,40.745,157.604
C07896=1033.551,-38.370,-84.704,168.248,40.746,157.604
C07897=1033.545,-38.620,-84.691,168.245,40.746,157.604
C07898=1033.539,-38.869,-84.678,168.243,40.747,157.604
C07899=1033.533,-39.119,-84.665,168.240,40.748,157.604
C07900=1033.526,-39.368,-84.653,168.238,40.749,157.604
C07901=1033.520,-39.618,-84.640,168.235,40.749,157.604
C07902=1033.513,-39.868,-84.627,168.232,40.750,157.604
C07903=1033.507,-40.118,-84.614,168.230,40.751,157.604
C07904=1033.500,-40.367,-84.601,168.228,40.752,157.604
C07905=1033.494,-40.617,-84.589,168.224,40.753,157.604
C07906=1033.488,-40.866,-84.576,168.223,40.753,157.604
C07907=1033.482,-41.116,-84.563,168.220,40.754,157.604
C07908=1033.475,-41.365,-84.550,168.217,40.755,157.604
C07909=1033.469,-41.615,-84.538,168.215,40.756,157.605
C07910=1033.463,-41.864,-84.524,168.212,40.757,157.604
C07911=1033.457,-42.114,-84.512,168.209,40.758,157.604
C07912=1033.451,-42.363,-84.500,168.207,40.759,157.605
C07913=1033.444,-42.613,-84.486,168.204,40.760,157.605
C07914=1033.438,-42.863,-84.474,168.202,40.760,157.605
C07915=1033.431,-43.113,-84.462,168.199,40.761,157.605
C07916=1033.425,-43.362,-84.449,168.196,40.762,157.605
C07917=1033.419,-43.612,-84.436,168.195,40.763,157.605
C07918=1033.413,-43.861,-84.423,168.192,40.764,157.605
C07919=1033.406,-44.111,-84.411,168.189,40.764,157.605
C07920=1033.400,-44.361,-84.398,168.187,40.765,157.605
C07921=1033.394,-44.610,-84.385,168.184,40.766,157.605
C07922=1033.388,-44.860,-84.372,168.181,40.767,157.605
C07923=1033.382,-45.109,-84.360,168.179,40.767,157.605
C07924=1033.375,-45.359,-84.347,168.176,40.768,157.605
C07925=1033.369,-45.608,-84.335,168.173,40.769,157.605
C07926=1033.363,-45.858,-84.323,168.171,40.770,157.605
C07927=1033.357,-46.108,-84.310,168.168,40.770,157.605
C07928=1033.351,-46.357,-84.297,168.165,40.771,157.605
C07929=1033.344,-46.607,-84.285,168.164,40.772,157.605
C07930=1033.338,-46.857,-84.272,168.161,40.773,157.605
C07931=1033.332,-47.107,-84.260,168.158,40.774,157.605
C07932=1033.326,-47.356,-84.246,168.156,40.774,157.605
C07933=1033.319,-47.605,-84.235,168.153,40.775,157.605
C07934=1033.313,-47.855,-84.222,168.150,40.776,157.605
C07935=1033.308,-48.104,-84.210,168.148,40.777,157.605
C07936=1033.301,-48.353,-84.197,168.145,40.777,157.605
C07937=1033.295,-48.603,-84.185,168.142,40.778,157.605
C07938=1033.289,-48.853,-84.172,168.140,40.779,157.605
C07939=1033.283,-49.103,-84.160,168.137,40.780,157.605
C07940=1033.277,-49.353,-84.147,168.134,40.781,157.605
C07941=1033.271,-49.602,-84.135,168.132,40.782,157.605
C07942=1033.264,-49.851,-84.122,168.130,40.783,157.605
C07943=1033.258,-50.101,-84.110,168.127,40.784,157.605
C07944=1033.252,-50.351,-84.097,168.125,40.784,157.605
C07945=1033.245,-50.601,-84.085,168.122,40.785,157.605
C07946=1033.240,-50.850,-84.073,168.119,40.786,157.605
C07947=1033.233,-51.100,-84.061,168.117,40.787,157.605
C07948=1033.227,-51.349,-84.049,168.114,40.788,157.605
C07949=1033.221,-51.599,-84.037,168.111,40.789,157.605
C07950=1033.213,-51.880,-84.023,168.108,40.790,157.605
C07951=1033.206,-52.161,-84.009,168.106,40.791,157.605
C07952=1033.199,-52.443,-83.996,168.103,40.792,157.605
C07953=1033.191,-52.725,-83.982,168.100,40.793,157.605
C07954=1033.186,-52.974,-83.970,168.097,40.794,157.606
C07955=1033.179,-53.223,-83.958,168.094,40.795,157.606
C07956=1033.173,-53.473,-83.946,168.091,40.796,157.606
C07957=1033.167,-53.723,-83.933,168.089,40.797,157.606
C07958=1033.160,-53.972,-83.921,168.086,40.798,157.606
C07959=1033.153,-54.222,-83.909,168.084,40.799,157.606
C07960=1033.148,-54.472,-83.897,168.081,40.800,157.606
C07961=1033.141,-54.722,-83.885,168.079,40.801,157.606
C07962=1033.135,-54.971,-83.874,168.076,40.802,157.606
C07963=1033.129,-55.221,-83.861,168.073,40.803,157.606
C07964=1033.123,-55.470,-83.849,168.070,40.804,157.606
C07965=1033.116,-55.720,-83.837,168.068,40.805,157.606
C07966=1033.109,-55.969,-83.825,168.065,40.806,157.606
C07967=1033.103,-56.219,-83.813,168.062,40.807,157.606
C07968=1033.098,-56.469,-83.802,168.060,40.808,157.606
C07969=1033.091,-56.718,-83.790,168.057,40.809,157.606
C07970=1033.085,-56.968,-83.777,168.055,40.810,157.606
C07971=1033.078,-57.218,-83.765,168.052,40.811,157.606
C07972=1033.072,-57.467,-83.754,168.049,40.812,157.606
C07973=1033.066,-57.717,-83.741,168.046,40.813,157.606
C07974=1033.060,-57.967,-83.730,168.044,40.814,157.606
C07975=1033.053,-58.216,-83.718,168.041,40.815,157.606
C07976=1033.047,-58.466,-83.706,168.039,40.816,157.606
C07977=1033.041,-58.716,-83.694,168.036,40.817,157.606
C07978=1033.035,-58.965,-83.683,168.034,40.818,157.607
C07979=1033.029,-59.215,-83.671,168.031,40.819,157.607
C07980=1033.022,-59.464,-83.659,168.028,40.820,157.607
C07981=1033.016,-59.714,-83.646,168.025,40.821,157.607
C07982=1033.010,-59.964,-83.635,168.022,40.822,157.607
C07983=1033.004,-60.213,-83.623,168.020,40.822,157.607
C07984=1032.998,-60.463,-83.611,168.017,40.823,157.607
C07985=1032.992,-60.712,-83.599,168.015,40.824,157.607
C07986=1032.985,-60.962,-83.588,168.012,40.825,157.607
C07987=1032.979,-61.212,-83.576,168.010,40.826,157.607
C07988=1032.973,-61.462,-83.564,168.007,40.827,157.607
C07989=1032.967,-61.711,-83.553,168.004,40.828,157.607
C07990=1032.960,-61.961,-83.541,168.001,40.829,157.607
C07991=1032.954,-62.210,-83.529,167.999,40.830,157.607
C07992=1032.949,-62.460,-83.517,167.996,40.831,157.607
C07993=1032.942,-62.710,-83.505,167.993,40.832,157.607
C07994=1032.935,-62.959,-83.493,167.991,40.833,157.607
C07995=1032.930,-63.209,-83.482,167.988,40.834,157.607
C07996=1032.924,-63.459,-83.470,167.986,40.835,157.607
C07997=1032.917,-63.709,-83.459,167.983,40.836,157.607
C07998=1032.911,-63.958,-83.447,167.980,40.837,157.607
C07999=1032.905,-64.207,-83.435,167.977,40.838,157.607
C08000=1032.899,-64.458,-83.423,167.974,40.839,157.607
C08001=1032.893,-64.707,-83.412,167.972,40.840,157.607
C08002=1032.887,-64.957,-83.400,167.970,40.841,157.607
C08003=1032.880,-65.207,-83.388,167.967,40.842,157.608
C08004=1032.874,-65.456,-83.378,167.964,40.843,157.608
C08005=1032.868,-65.706,-83.365,167.962,40.844,157.608
C08006=1032.862,-65.955,-83.353,167.959,40.845,157.608
C08007=1032.856,-66.205,-83.342,167.956,40.846,157.608
C08008=1032.849,-66.455,-83.330,167.953,40.847,157.608
C08009=1032.844,-66.704,-83.319,167.950,40.848,157.608
C08010=1032.838,-66.954,-83.307,167.948,40.849,157.608
C08011=1032.832,-67.203,-83.296,167.946,40.850,157.608
C08012=1032.825,-67.453,-83.284,167.943,40.851,157.608
C08013=1032.820,-67.702,-83.273,167.940,40.852,157.608
C08014=1032.813,-67.985,-83.260,167.937,40.853,157.608
C08015=1032.806,-68.269,-83.247,167.934,40.854,157.608
C08016=1032.799,-68.551,-83.234,167.931,40.855,157.608
C08017=1032.792,-68.834,-83.221,167.928,40.856,157.608
C08018=1032.786,-69.083,-83.209,167.925,40.857,157.608
C08019=1032.780,-69.333,-83.197,167.923,40.858,157.608
C08020=1032.774,-69.582,-83.186,167.920,40.859,157.608
C08021=1032.768,-69.832,-83.175,167.917,40.860,157.608
C08022=1032.762,-70.082,-83.164,167.915,40.861,157.608
C08023=1032.756,-70.331,-83.152,167.912,40.862,157.608
C08024=1032.751,-70.581,-83.140,167.909,40.863,157.608
C08025=1032.744,-70.831,-83.128,167.906,40.864,157.608
C08026=1032.738,-71.080,-83.117,167.903,40.865,157.608
C08027=1032.732,-71.330,-83.106,167.902,40.866,157.609
C08028=1032.726,-71.579,-83.095,167.899,40.867,157.609
C08029=1032.720,-71.829,-83.083,167.896,40.868,157.609
C08030=1032.715,-72.079,-83.072,167.893,40.869,157.609
C08031=1032.708,-72.329,-83.060,167.890,40.870,157.609
C08032=1032.702,-72.578,-83.049,167.888,40.871,157.609
C08033=1032.696,-72.828,-83.038,167.885,40.872,157.609
C08034=1032.690,-73.078,-83.027,167.882,40.873,157.609
C08035=1032.685,-73.327,-83.015,167.879,40.874,157.609
C08036=1032.678,-73.577,-83.003,167.877,40.875,157.609
C08037=1032.673,-73.827,-82.993,167.874,40.876,157.609
C08038=1032.666,-74.076,-82.981,167.872,40.877,157.609
C08039=1032.660,-74.326,-82.970,167.869,40.879,157.609
C08040=1032.655,-74.575,-82.959,167.866,40.880,157.609
C08041=1032.648,-74.826,-82.948,167.863,40.881,157.609
C08042=1032.643,-75.075,-82.937,167.860,40.882,157.609
C08043=1032.636,-75.325,-82.925,167.857,40.883,157.609
C08044=1032.630,-75.574,-82.914,167.855,40.884,157.609
///RCONF 1,0,0,1,0,0,0,0,0,0,0,0,0,0,0,0,0,0,0,0,0,0,0,0
C08045=1032.623,-75.824,-82.903,167.853,40.885,157.609
C08046=1032.617,-76.074,-82.892,167.850,40.886,157.609
C08047=1032.612,-76.323,-82.881,167.847,40.887,157.609
C08048=1032.605,-76.573,-82.870,167.844,40.889,157.610
C08049=1032.599,-76.823,-82.859,167.841,40.890,157.610
C08050=1032.593,-77.073,-82.848,167.839,40.891,157.610
C08051=1032.587,-77.322,-82.837,167.836,40.892,157.610
C08052=1032.582,-77.572,-82.826,167.834,40.893,157.610
C08053=1032.575,-77.822,-82.815,167.831,40.895,157.610
C08054=1032.569,-78.071,-82.805,167.828,40.896,157.610
C08055=1032.563,-78.321,-82.794,167.825,40.897,157.610
C08056=1032.556,-78.570,-82.782,167.822,40.898,157.610
C08057=1032.551,-78.820,-82.771,167.820,40.899,157.610
C08058=1032.544,-79.070,-82.760,167.817,40.900,157.610
C08059=1032.539,-79.319,-82.749,167.814,40.901,157.610
C08060=1032.533,-79.569,-82.738,167.811,40.902,157.610
C08061=1032.527,-79.819,-82.727,167.809,40.903,157.610
C08062=1032.520,-80.068,-82.717,167.806,40.905,157.610
C08063=1032.515,-80.318,-82.706,167.804,40.906,157.611
C08064=1032.508,-80.569,-82.695,167.801,40.907,157.611
C08065=1032.502,-80.818,-82.685,167.798,40.909,157.611
C08066=1032.496,-81.067,-82.674,167.795,40.910,157.611
C08067=1032.489,-81.317,-82.663,167.792,40.911,157.611
C08068=1032.483,-81.567,-82.652,167.789,40.912,157.611
C08069=1032.478,-81.816,-82.642,167.787,40.913,157.611
C08070=1032.470,-82.066,-82.631,167.784,40.915,157.611
C08071=1032.465,-82.316,-82.621,167.781,40.916,157.611
C08072=1032.459,-82.566,-82.610,167.778,40.918,157.611
C08073=1032.452,-82.816,-82.599,167.775,40.919,157.611
///RCONF 1,0,0,0,0,0,0,0,0,0,0,0,0,0,0,0,0,0,0,0,0,0,0,0
C08074=1032.446,-83.065,-82.588,167.773,40.920,157.611
C08075=1032.440,-83.314,-82.578,167.771,40.921,157.612
C08076=1032.434,-83.564,-82.567,167.768,40.922,157.612
C08077=1032.428,-83.815,-82.557,167.765,40.924,157.612
C08078=1032.421,-84.099,-82.544,167.761,40.925,157.612
C08079=1032.414,-84.384,-82.532,167.758,40.927,157.612
C08080=1032.406,-84.668,-82.520,167.756,40.928,157.612
C08081=1032.400,-84.953,-82.508,167.752,40.929,157.612
C08082=1032.394,-85.202,-82.498,167.749,40.931,157.612
C08083=1032.388,-85.453,-82.487,167.746,40.932,157.612
C08084=1032.381,-85.702,-82.477,167.743,40.933,157.612
C08085=1032.376,-85.952,-82.466,167.742,40.935,157.612
C08086=1032.369,-86.202,-82.456,167.739,40.936,157.612
C08087=1032.364,-86.451,-82.445,167.736,40.937,157.612
C08088=1032.357,-86.701,-82.434,167.733,40.938,157.613
C08089=1032.351,-86.950,-82.424,167.730,40.939,157.613
C08090=1032.346,-87.201,-82.414,167.727,40.941,157.613
C08091=1032.339,-87.450,-82.404,167.724,40.942,157.613
C08092=1032.333,-87.700,-82.392,167.722,40.944,157.613
C08093=1032.327,-87.950,-82.383,167.719,40.945,157.613
C08094=1032.321,-88.199,-82.372,167.716,40.946,157.613
C08095=1032.315,-88.449,-82.361,167.713,40.948,157.613
C08096=1032.309,-88.699,-82.351,167.710,40.949,157.613
C08097=1032.303,-88.948,-82.340,167.708,40.950,157.613
C08098=1032.296,-89.199,-82.331,167.705,40.951,157.613
C08099=1032.291,-89.448,-82.320,167.702,40.952,157.613
C08100=1032.284,-89.697,-82.309,167.699,40.954,157.614
C08101=1032.279,-89.947,-82.299,167.696,40.955,157.614
C08102=1032.273,-90.197,-82.288,167.693,40.957,157.614
C08103=1032.267,-90.447,-82.279,167.691,40.958,157.614
C08104=1032.261,-90.696,-82.268,167.689,40.959,157.614
C08105=1032.255,-90.945,-82.258,167.686,40.960,157.614
C08106=1032.249,-91.196,-82.247,167.683,40.961,157.614
C08107=1032.242,-91.445,-82.237,167.680,40.963,157.614
C08108=1032.237,-91.695,-82.227,167.677,40.964,157.614
C08109=1032.231,-91.945,-82.216,167.675,40.966,157.614
C08110=1032.225,-92.195,-82.206,167.672,40.967,157.614
C08111=1032.219,-92.444,-82.195,167.669,40.968,157.615
C08112=1032.213,-92.694,-82.186,167.666,40.969,157.615
C08113=1032.207,-92.943,-82.175,167.663,40.970,157.615
C08114=1032.201,-93.193,-82.165,167.661,40.972,157.615
C08115=1032.195,-93.443,-82.154,167.658,40.973,157.615
C08116=1032.189,-93.693,-82.145,167.655,40.975,157.615
C08117=1032.183,-93.942,-82.134,167.652,40.976,157.615
C08118=1032.177,-94.192,-82.124,167.649,40.977,157.615
C08119=1032.172,-94.442,-82.114,167.646,40.978,157.615
C08120=1032.165,-94.692,-82.104,167.644,40.979,157.615
C08121=1032.159,-94.942,-82.093,167.641,40.981,157.615
C08122=1032.153,-95.191,-82.083,167.638,40.982,157.615
C08123=1032.147,-95.441,-82.073,167.635,40.984,157.615
C08124=1032.142,-95.691,-82.063,167.632,40.985,157.615
C08125=1032.135,-95.940,-82.053,167.630,40.987,157.616
C08126=1032.130,-96.191,-82.042,167.628,40.987,157.616
C08127=1032.123,-96.440,-82.032,167.625,40.989,157.616
C08128=1032.118,-96.690,-82.022,167.622,40.990,157.616
C08129=1032.112,-96.939,-82.013,167.619,40.991,157.616
C08130=1032.107,-97.188,-82.002,167.616,40.993,157.616
C08131=1032.100,-97.438,-81.992,167.614,40.994,157.616
C08132=1032.095,-97.688,-81.982,167.611,40.996,157.616
C08133=1032.089,-97.938,-81.973,167.608,40.997,157.616
C08134=1032.082,-98.187,-81.962,167.605,40.998,157.616
C08135=1032.076,-98.437,-81.953,167.603,41.000,157.617
C08136=1032.071,-98.687,-81.943,167.600,41.001,157.617
C08137=1032.065,-98.937,-81.933,167.597,41.003,157.617
C08138=1032.058,-99.186,-81.923,167.594,41.004,157.617
C08139=1032.052,-99.436,-81.913,167.591,41.005,157.617
C08140=1032.047,-99.686,-81.903,167.589,41.007,157.617
C08141=1032.040,-99.936,-81.893,167.586,41.009,157.617
C08142=1032.034,-100.203,-81.883,167.582,41.010,157.617
C08143=1032.027,-100.469,-81.873,167.579,41.012,157.617
C08144=1032.021,-100.736,-81.861,167.576,41.013,157.617
C08145=1032.015,-101.002,-81.851,167.574,41.015,157.618
C08146=1032.009,-101.252,-81.841,167.571,41.016,157.618
C08147=1032.002,-101.502,-81.832,167.568,41.018,157.618
C08148=1031.997,-101.752,-81.822,167.565,41.019,157.618
C08149=1031.991,-102.002,-81.812,167.562,41.020,157.618
C08150=1031.984,-102.272,-81.802,167.559,41.022,157.618
C08151=1031.977,-102.542,-81.791,167.556,41.024,157.618
C08152=1031.971,-102.812,-81.781,167.553,41.025,157.618
C08153=1031.965,-103.082,-81.769,167.550,41.027,157.618
C08154=1031.959,-103.331,-81.760,167.548,41.028,157.619
C08155=1031.953,-103.581,-81.751,167.544,41.030,157.619
C08156=1031.947,-103.831,-81.741,167.541,41.031,157.619
C08157=1031.941,-104.081,-81.731,167.538,41.033,157.619
C08158=1031.935,-104.330,-81.721,167.536,41.035,157.619
C08159=1031.929,-104.580,-81.712,167.533,41.036,157.619
C08160=1031.923,-104.830,-81.702,167.530,41.037,157.619
C08161=1031.917,-105.079,-81.693,167.527,41.039,157.619
C08162=1031.912,-105.329,-81.683,167.524,41.040,157.619
C08163=1031.906,-105.579,-81.673,167.522,41.042,157.620
C08164=1031.899,-105.829,-81.664,167.519,41.043,157.620
C08165=1031.893,-106.079,-81.654,167.516,41.044,157.620
C08166=1031.888,-106.328,-81.645,167.513,41.046,157.620
C08167=1031.881,-106.578,-81.635,167.510,41.048,157.620
C08168=1031.876,-106.828,-81.625,167.508,41.049,157.620
C08169=1031.870,-107.078,-81.616,167.505,41.051,157.620
C08170=1031.864,-107.328,-81.607,167.502,41.052,157.620
C08171=1031.858,-107.577,-81.598,167.499,41.054,157.620
C08172=1031.852,-107.827,-81.588,167.496,41.055,157.620
C08173=1031.846,-108.077,-81.579,167.494,41.057,157.621
C08174=1031.840,-108.326,-81.569,167.491,41.058,157.621
C08175=1031.834,-108.576,-81.559,167.488,41.060,157.621
C08176=1031.828,-108.825,-81.550,167.486,41.062,157.621
C08177=1031.822,-109.076,-81.541,167.483,41.063,157.621
C08178=1031.816,-109.325,-81.532,167.480,41.064,157.621
C08179=1031.810,-109.575,-81.522,167.476,41.066,157.621
C08180=1031.804,-109.824,-81.513,167.473,41.068,157.621
C08181=1031.798,-110.074,-81.503,167.471,41.070,157.622
C08182=1031.792,-110.325,-81.495,167.468,41.071,157.622
C08183=1031.786,-110.574,-81.485,167.465,41.072,157.622
C08184=1031.781,-110.823,-81.476,167.462,41.074,157.622
C08185=1031.774,-111.073,-81.466,167.460,41.076,157.622
C08186=1031.769,-111.324,-81.457,167.457,41.077,157.622
C08187=1031.762,-111.574,-81.448,167.454,41.079,157.622
C08188=1031.757,-111.823,-81.439,167.451,41.080,157.622
C08189=1031.751,-112.072,-81.429,167.449,41.082,157.623
C08190=1031.745,-112.323,-81.420,167.446,41.084,157.623
C08191=1031.739,-112.572,-81.411,167.443,41.085,157.623
C08192=1031.733,-112.822,-81.401,167.440,41.087,157.623
C08193=1031.727,-113.072,-81.393,167.437,41.088,157.623
C08194=1031.722,-113.321,-81.383,167.434,41.090,157.623
C08195=1031.715,-113.571,-81.374,167.431,41.092,157.623
C08196=1031.709,-113.821,-81.364,167.428,41.093,157.623
C08197=1031.704,-114.071,-81.356,167.426,41.095,157.624
C08198=1031.698,-114.320,-81.346,167.423,41.097,157.624
C08199=1031.692,-114.571,-81.337,167.420,41.098,157.624
C08200=1031.686,-114.820,-81.328,167.417,41.099,157.624
C08201=1031.680,-115.070,-81.319,167.414,41.101,157.624
C08202=1031.674,-115.320,-81.310,167.412,41.103,157.624
C08203=1031.669,-115.569,-81.301,167.409,41.105,157.624
C08204=1031.663,-115.820,-81.292,167.406,41.106,157.624
C08205=1031.657,-116.068,-81.283,167.403,41.108,157.625
C08206=1031.650,-116.355,-81.272,167.400,41.110,157.625
C08207=1031.643,-116.642,-81.262,167.396,41.112,157.625
C08208=1031.636,-116.928,-81.252,167.393,41.113,157.625
C08209=1031.630,-117.214,-81.241,167.390,41.116,157.625
C08210=1031.624,-117.465,-81.232,167.387,41.117,157.625
C08211=1031.618,-117.714,-81.224,167.384,41.119,157.625
C08212=1031.612,-117.964,-81.215,167.381,41.120,157.626
C08213=1031.606,-118.214,-81.205,167.379,41.122,157.626
C08214=1031.600,-118.464,-81.197,167.376,41.124,157.626
C08215=1031.594,-118.713,-81.187,167.373,41.125,157.626
C08216=1031.589,-118.963,-81.179,167.370,41.127,157.626
C08217=1031.582,-119.213,-81.170,167.368,41.129,157.626
C08218=1031.577,-119.462,-81.161,167.364,41.131,157.626
C08219=1031.571,-119.712,-81.152,167.361,41.132,157.626
C08220=1031.565,-119.962,-81.143,167.358,41.134,157.627
C08221=1031.560,-120.212,-81.135,167.356,41.136,157.627
C08222=1031.553,-120.462,-81.126,167.353,41.137,157.627
C08223=1031.547,-120.711,-81.117,167.350,41.139,157.627
C08224=1031.541,-120.961,-81.107,167.348,41.141,157.627
C08225=1031.536,-121.211,-81.099,167.345,41.143,157.627
C08226=1031.529,-121.461,-81.091,167.342,41.144,157.627
C08227=1031.524,-121.710,-81.082,167.339,41.146,157.628
C08228=1031.518,-121.961,-81.073,167.336,41.148,157.628
C08229=1031.513,-122.210,-81.064,167.333,41.149,157.628
C08230=1031.506,-122.460,-81.055,167.330,41.151,157.628
C08231=1031.500,-122.709,-81.047,167.327,41.153,157.628
C08232=1031.495,-122.960,-81.038,167.325,41.155,157.628
C08233=1031.489,-123.209,-81.029,167.322,41.156,157.628
C08234=1031.482,-123.459,-81.020,167.319,41.158,157.629
C08235=1031.477,-123.709,-81.012,167.316,41.160,157.629
C08236=1031.472,-123.958,-81.003,167.314,41.161,157.629
C08237=1031.466,-124.208,-80.994,167.310,41.163,157.629
C08238=1031.460,-124.458,-80.986,167.307,41.165,157.629
C08239=1031.454,-124.708,-80.977,167.305,41.167,157.629
C08240=1031.449,-124.958,-80.969,167.302,41.168,157.629
C08241=1031.442,-125.207,-80.960,167.299,41.171,157.630
C08242=1031.436,-125.457,-80.951,167.296,41.173,157.630
C08243=1031.430,-125.707,-80.943,167.294,41.174,157.630
C08244=1031.425,-125.957,-80.934,167.291,41.176,157.630
C08245=1031.419,-126.207,-80.926,167.287,41.178,157.630
C08246=1031.413,-126.457,-80.918,167.285,41.179,157.630
C08247=1031.407,-126.706,-80.909,167.282,41.181,157.631
C08248=1031.400,-126.956,-80.900,167.279,41.183,157.631
C08249=1031.395,-127.206,-80.892,167.276,41.185,157.631
C08250=1031.390,-127.455,-80.883,167.274,41.187,157.631
C08251=1031.384,-127.705,-80.875,167.271,41.189,157.631
C08252=1031.378,-127.954,-80.866,167.267,41.191,157.631
C08253=1031.373,-128.204,-80.857,167.265,41.191,157.631
C08254=1031.368,-128.454,-80.847,167.263,41.193,157.631
C08255=1031.365,-128.703,-80.837,167.259,41.193,157.631
C08256=1031.362,-128.953,-80.826,167.257,41.192,157.631
C08257=1031.360,-129.203,-80.815,167.255,41.192,157.631
C08258=1031.357,-129.453,-80.803,167.253,41.191,157.631
C08259=1031.356,-129.703,-80.790,167.250,41.190,157.630
C08260=1031.355,-129.952,-80.777,167.249,41.187,157.630
C08261=1031.355,-130.202,-80.763,167.246,41.185,157.629
C08262=1031.357,-130.453,-80.748,167.244,41.182,157.629
C08263=1031.357,-130.702,-80.734,167.243,41.179,157.628
C08264=1031.360,-130.953,-80.718,167.242,41.175,157.627
C08265=1031.362,-131.202,-80.702,167.240,41.171,157.626
C08266=1031.366,-131.452,-80.685,167.239,41.166,157.626
C08267=1031.370,-131.703,-80.668,167.237,41.160,157.625
C08268=1031.374,-131.952,-80.650,167.236,41.155,157.624
C08269=1031.380,-132.202,-80.631,167.235,41.149,157.623
C08270=1031.057,-132.227,-80.929,167.185,41.384,157.659
C08271=1031.051,-131.977,-80.947,167.187,41.390,157.660
C08272=1031.047,-131.727,-80.966,167.188,41.396,157.661
C08273=1031.043,-131.477,-80.983,167.189,41.401,157.662
C08274=1031.040,-131.227,-80.999,167.190,41.406,157.663
C08275=1031.037,-130.977,-81.016,167.192,41.410,157.664
C08276=1031.035,-130.727,-81.031,167.194,41.414,157.665
C08277=1031.033,-130.477,-81.046,167.196,41.417,157.665
C08278=1031.033,-130.227,-81.060,167.198,41.421,157.666
C08279=1031.033,-129.978,-81.075,167.200,41.423,157.666
C08280=1031.033,-129.728,-81.088,167.202,41.425,157.667
C08281=1031.034,-129.478,-81.101,167.204,41.426,157.667
C08282=1031.037,-129.228,-81.113,167.206,41.428,157.668
C08283=1031.039,-128.978,-81.124,167.208,41.428,157.668
C08284=1031.042,-128.728,-81.135,167.211,41.428,157.668
C08285=1031.046,-128.479,-81.145,167.213,41.428,157.668
C08286=1031.050,-128.230,-81.156,167.216,41.427,157.668
C08287=1031.054,-127.980,-81.165,167.219,41.426,157.668
C08288=1031.060,-127.730,-81.173,167.222,41.424,157.668
C08289=1031.066,-127.480,-81.181,167.225,41.423,157.668
C08290=1031.073,-127.231,-81.190,167.227,41.420,157.668
C08291=1031.078,-126.981,-81.199,167.230,41.418,157.667
C08292=1031.084,-126.731,-81.207,167.234,41.417,157.667
C08293=1031.090,-126.481,-81.215,167.236,41.415,157.667
C08294=1031.095,-126.232,-81.224,167.239,41.413,157.667
C08295=1031.102,-125.982,-81.232,167.242,41.411,157.667
C08296=1031.107,-125.732,-81.241,167.244,41.409,157.667
C08297=1031.113,-125.482,-81.250,167.247,41.407,157.667
C08298=1031.119,-125.233,-81.258,167.250,41.405,157.666
C08299=1031.125,-124.982,-81.267,167.254,41.404,157.666
C08300=1031.131,-124.733,-81.275,167.256,41.402,157.666
C08301=1031.136,-124.484,-81.284,167.259,41.400,157.666
C08302=1031.142,-124.233,-81.293,167.262,41.398,157.666
C08303=1031.148,-123.984,-81.301,167.265,41.397,157.666
C08304=1031.154,-123.733,-81.310,167.267,41.394,157.665
C08305=1031.160,-123.484,-81.319,167.271,41.392,157.665
C08306=1031.166,-123.234,-81.328,167.274,41.391,157.665
C08307=1031.172,-122.985,-81.335,167.276,41.389,157.665
C08308=1031.177,-122.734,-81.344,167.279,41.387,157.665
C08309=1031.183,-122.485,-81.354,167.282,41.386,157.665
C08310=1031.188,-122.235,-81.362,167.284,41.384,157.665
C08311=1031.195,-121.985,-81.370,167.287,41.382,157.665
C08312=1031.200,-121.736,-81.379,167.290,41.380,157.664
C08313=1031.206,-121.486,-81.388,167.294,41.378,157.664
C08314=1031.212,-121.236,-81.397,167.296,41.377,157.664
C08315=1031.218,-120.987,-81.406,167.299,41.375,157.664
C08316=1031.224,-120.737,-81.414,167.302,41.373,157.664
C08317=1031.230,-120.486,-81.423,167.305,41.372,157.664
C08318=1031.235,-120.237,-81.432,167.307,41.370,157.664
C08319=1031.241,-119.987,-81.441,167.310,41.368,157.663
C08320=1031.248,-119.737,-81.450,167.313,41.366,157.663
C08321=1031.253,-119.488,-81.459,167.316,41.365,157.663
C08322=1031.259,-119.237,-81.467,167.319,41.363,157.663
C08323=1031.265,-118.988,-81.477,167.322,41.361,157.663
C08324=1031.271,-118.738,-81.485,167.325,41.359,157.663
C08325=1031.277,-118.489,-81.494,167.327,41.358,157.663
C08326=1031.283,-118.239,-81.503,167.330,41.356,157.663
C08327=1031.288,-117.989,-81.512,167.333,41.354,157.662
C08328=1031.294,-117.739,-81.521,167.336,41.352,157.662
C08329=1031.300,-117.489,-81.531,167.339,41.351,157.662
C08330=1031.306,-117.240,-81.539,167.342,41.349,157.662
C08331=1031.313,-116.953,-81.549,167.345,41.347,157.662
C08332=1031.319,-116.667,-81.560,167.348,41.345,157.662
C08333=1031.326,-116.380,-81.569,167.351,41.343,157.661
C08334=1031.333,-116.094,-81.580,167.355,41.341,157.661
C08335=1031.339,-115.845,-81.590,167.357,41.339,157.661
C08336=1031.344,-115.594,-81.598,167.360,41.338,157.661
C08337=1031.351,-115.345,-81.607,167.363,41.336,157.661
C08338=1031.357,-115.095,-81.616,167.366,41.334,157.661
C08339=1031.363,-114.845,-81.625,167.369,41.332,157.661
C08340=1031.369,-114.595,-81.634,167.372,41.331,157.661
C08341=1031.374,-114.346,-81.643,167.375,41.329,157.660
C08342=1031.380,-114.096,-81.653,167.378,41.327,157.660
C08343=1031.386,-113.846,-81.662,167.380,41.325,157.660
C08344=1031.392,-113.596,-81.671,167.383,41.324,157.660
C08345=1031.398,-113.347,-81.681,167.386,41.323,157.660
C08346=1031.404,-113.096,-81.689,167.389,41.321,157.660
C08347=1031.409,-112.847,-81.699,167.391,41.319,157.660
C08348=1031.416,-112.597,-81.708,167.394,41.318,157.660
C08349=1031.421,-112.347,-81.717,167.398,41.316,157.659
C08350=1031.427,-112.098,-81.726,167.401,41.314,157.659
C08351=1031.433,-111.848,-81.736,167.403,41.312,157.659
C08352=1031.439,-111.598,-81.745,167.406,41.311,157.659
C08353=1031.445,-111.349,-81.754,167.409,41.309,157.659
C08354=1031.451,-111.099,-81.763,167.412,41.308,157.659
C08355=1031.457,-110.849,-81.773,167.414,41.306,157.659
C08356=1031.462,-110.599,-81.782,167.417,41.304,157.659
C08357=1031.468,-110.349,-81.791,167.420,41.303,157.658
C08358=1031.475,-110.100,-81.801,167.422,41.301,157.658
C08359=1031.481,-109.850,-81.810,167.425,41.299,157.658
C08360=1031.486,-109.601,-81.819,167.429,41.298,157.658
C08361=1031.492,-109.350,-81.828,167.432,41.296,157.658
C08362=1031.498,-109.100,-81.838,167.435,41.295,157.658
C08363=1031.505,-108.851,-81.847,167.437,41.293,157.658
C08364=1031.510,-108.602,-81.857,167.440,41.291,157.658
C08365=1031.516,-108.352,-81.866,167.443,41.289,157.657
C08366=1031.522,-108.101,-81.875,167.445,41.288,157.657
C08367=1031.528,-107.852,-81.885,167.448,41.287,157.657
C08368=1031.534,-107.602,-81.894,167.451,41.285,157.657
C08369=1031.540,-107.353,-81.903,167.454,41.283,157.657
C08370=1031.546,-107.103,-81.913,167.457,41.282,157.657
C08371=1031.552,-106.853,-81.923,167.459,41.280,157.657
C08372=1031.558,-106.603,-81.933,167.463,41.279,157.657
C08373=1031.563,-106.354,-81.942,167.466,41.277,157.657
C08374=1031.570,-106.104,-81.951,167.469,41.275,157.656
C08375=1031.576,-105.854,-81.961,167.471,41.273,157.656
C08376=1031.582,-105.604,-81.971,167.474,41.272,157.656
C08377=1031.588,-105.354,-81.979,167.477,41.271,157.656
C08378=1031.593,-105.105,-81.989,167.480,41.269,157.656
C08379=1031.599,-104.855,-81.999,167.482,41.267,157.656
C08380=1031.605,-104.605,-82.008,167.485,41.266,157.656
C08381=1031.611,-104.355,-82.018,167.488,41.265,157.656
C08382=1031.617,-104.105,-82.027,167.491,41.263,157.656
C08383=1031.623,-103.855,-82.038,167.494,41.262,157.656
C08384=1031.629,-103.607,-82.048,167.496,41.260,157.655
C08385=1031.635,-103.357,-82.057,167.499,41.258,157.655
C08386=1031.641,-103.107,-82.067,167.502,41.257,157.655
C08387=1031.647,-102.858,-82.076,167.505,41.256,157.655
C08388=1031.653,-102.607,-82.086,167.507,41.254,157.655
C08389=1031.659,-102.358,-82.096,167.510,41.252,157.655
C08390=1031.665,-102.108,-82.106,167.513,41.251,157.655
C08391=1031.671,-101.858,-82.115,167.517,41.249,157.655
C08392=1031.676,-101.609,-82.125,167.519,41.248,157.654
C08393=1031.682,-101.359,-82.134,167.522,41.247,157.654
C08394=1031.688,-101.109,-82.144,167.525,41.245,157.654
C08395=1031.696,-100.822,-82.155,167.528,41.243,157.654
C08396=1031.702,-100.535,-82.167,167.532,41.241,157.654
C08397=1031.709,-100.248,-82.179,167.534,41.240,157.654
C08398=1031.716,-99.961,-82.190,167.538,41.238,157.654
C08399=1031.722,-99.712,-82.199,167.541,41.236,157.654
C08400=1031.728,-99.462,-82.209,167.544,41.235,157.654
C08401=1031.734,-99.212,-82.219,167.546,41.233,157.653
C08402=1031.740,-98.963,-82.229,167.549,41.232,157.653
C08403=1031.746,-98.713,-82.239,167.552,41.231,157.653
C08404=1031.752,-98.463,-82.249,167.555,41.229,157.653
C08405=1031.758,-98.213,-82.258,167.557,41.227,157.653
C08406=1031.764,-97.963,-82.268,167.560,41.226,157.653
C08407=1031.771,-97.714,-82.278,167.563,41.224,157.653
C08408=1031.776,-97.464,-82.288,167.566,41.223,157.653
C08409=1031.782,-97.214,-82.298,167.569,41.222,157.653
C08410=1031.788,-96.964,-82.309,167.571,41.220,157.653
C08411=1031.794,-96.715,-82.318,167.574,41.219,157.653
C08412=1031.799,-96.465,-82.329,167.577,41.217,157.652
C08413=1031.806,-96.215,-82.339,167.580,41.216,157.652
C08414=1031.811,-95.965,-82.349,167.583,41.215,157.652
C08415=1031.818,-95.715,-82.359,167.586,41.213,157.652
C08416=1031.823,-95.466,-82.370,167.588,41.212,157.652
C08417=1031.829,-95.216,-82.379,167.591,41.211,157.652
C08418=1031.835,-94.966,-82.389,167.594,41.209,157.652
C08419=1031.841,-94.717,-82.400,167.597,41.208,157.652
C08420=1031.847,-94.467,-82.410,167.599,41.206,157.652
C08421=1031.853,-94.218,-82.420,167.602,41.205,157.652
C08422=1031.859,-93.968,-82.430,167.605,41.204,157.652
C08423=1031.864,-93.718,-82.441,167.608,41.203,157.652
C08424=1031.871,-93.468,-82.451,167.611,41.201,157.651
C08425=1031.876,-93.218,-82.461,167.614,41.200,157.651
C08426=1031.883,-92.969,-82.471,167.616,41.198,157.651
C08427=1031.888,-92.719,-82.481,167.619,41.197,157.651
C08428=1031.894,-92.470,-82.491,167.622,41.195,157.651
C08429=1031.900,-92.220,-82.502,167.625,41.194,157.651
C08430=1031.906,-91.970,-82.512,167.628,41.193,157.651
C08431=1031.912,-91.720,-82.522,167.630,41.192,157.651
C08432=1031.918,-91.471,-82.532,167.633,41.191,157.651
C08433=1031.924,-91.220,-82.543,167.636,41.189,157.651
C08434=1031.931,-90.971,-82.553,167.639,41.188,157.651
C08435=1031.937,-90.722,-82.564,167.642,41.186,157.651
C08436=1031.942,-90.471,-82.574,167.645,41.185,157.650
C08437=1031.948,-90.222,-82.585,167.647,41.183,157.650
C08438=1031.954,-89.972,-82.595,167.649,41.182,157.650
C08439=1031.960,-89.723,-82.605,167.652,41.181,157.650
C08440=1031.966,-89.473,-82.615,167.655,41.180,157.650
C08441=1031.973,-89.223,-82.626,167.657,41.178,157.650
C08442=1031.979,-88.974,-82.637,167.660,41.177,157.650
C08443=1031.984,-88.723,-82.647,167.663,41.175,157.650
C08444=1031.991,-88.474,-82.657,167.666,41.174,157.650
C08445=1031.996,-88.224,-82.667,167.669,41.173,157.650
C08446=1032.002,-87.975,-82.678,167.672,41.172,157.650
C08447=1032.009,-87.725,-82.689,167.674,41.170,157.649
C08448=1032.015,-87.475,-82.698,167.677,41.169,157.649
C08449=1032.021,-87.225,-82.709,167.680,41.167,157.649
C08450=1032.026,-86.976,-82.720,167.683,41.166,157.649
C08451=1032.036,-86.630,-82.734,167.687,41.164,157.649
C08452=1032.043,-86.284,-82.748,167.690,41.162,157.649
C08453=1032.052,-85.938,-82.763,167.695,41.161,157.649
C08454=1032.061,-85.592,-82.778,167.699,41.159,157.649
C08455=1032.066,-85.373,-82.787,167.700,41.157,157.649
C08456=1032.071,-85.154,-82.797,167.703,41.156,157.649
C08457=1032.077,-84.935,-82.805,167.705,41.155,157.649
C08458=1032.082,-84.715,-82.815,167.708,41.154,157.649
C08459=1032.087,-84.497,-82.824,167.711,41.152,157.648
C08460=1032.092,-84.277,-82.834,167.713,41.152,157.648
C08461=1032.098,-84.059,-82.842,167.716,41.151,157.648
C08462=1032.103,-83.839,-82.852,167.717,41.149,157.648
C08463=1032.109,-83.590,-82.863,167.720,41.148,157.648
C08464=1032.115,-83.340,-82.873,167.723,41.147,157.648
C08465=1032.122,-83.090,-82.884,167.726,41.145,157.648
C08466=1032.128,-82.841,-82.894,167.729,41.144,157.648
C08467=1032.134,-82.591,-82.905,167.731,41.142,157.648
C08468=1032.140,-82.341,-82.916,167.734,41.141,157.648
C08469=1032.146,-82.091,-82.926,167.737,41.140,157.648
C08470=1032.152,-81.842,-82.937,167.740,41.139,157.648
C08471=1032.158,-81.592,-82.948,167.743,41.137,157.647
C08472=1032.165,-81.342,-82.958,167.746,41.136,157.647
C08473=1032.171,-81.093,-82.969,167.748,41.134,157.647
C08474=1032.178,-80.843,-82.980,167.751,41.133,157.647
C08475=1032.183,-80.594,-82.991,167.754,41.132,157.647
C08476=1032.189,-80.344,-83.001,167.757,41.131,157.647
C08477=1032.196,-80.094,-83.011,167.760,41.130,157.647
C08478=1032.202,-79.844,-83.022,167.762,41.128,157.647
C08479=1032.207,-79.595,-83.033,167.765,41.127,157.647
C08480=1032.214,-79.344,-83.044,167.768,41.126,157.647
C08481=1032.220,-79.095,-83.055,167.771,41.124,157.647
C08482=1032.225,-78.845,-83.066,167.773,41.123,157.647
C08483=1032.232,-78.596,-83.077,167.776,41.122,157.647
C08484=1032.238,-78.346,-83.088,167.778,41.120,157.646
C08485=1032.244,-78.097,-83.099,167.781,41.119,157.646
C08486=1032.250,-77.846,-83.110,167.784,41.118,157.646
C08487=1032.256,-77.597,-83.121,167.787,41.117,157.646
C08488=1032.262,-77.348,-83.132,167.790,41.116,157.646
C08489=1032.268,-77.098,-83.144,167.793,41.115,157.646
C08490=1032.274,-76.848,-83.154,167.796,41.114,157.646
C08491=1032.281,-76.598,-83.165,167.798,41.113,157.646
C08492=1032.287,-76.349,-83.176,167.800,41.111,157.646
C08493=1032.293,-76.099,-83.187,167.803,41.110,157.646
C08494=1032.299,-75.849,-83.198,167.806,41.109,157.646
C08495=1032.305,-75.600,-83.209,167.809,41.107,157.646
C08496=1032.311,-75.350,-83.220,167.812,41.106,157.646
///RCONF 1,0,0,1,0,0,0,0,0,0,0,0,0,0,0,0,0,0,0,0,0,0,0,0
C08497=1032.317,-75.100,-83.231,167.814,41.105,157.646
C08498=1032.323,-74.851,-83.243,167.817,41.104,157.646
C08499=1032.329,-74.601,-83.254,167.820,41.103,157.645
C08500=1032.335,-74.352,-83.265,167.823,41.102,157.645
C08501=1032.342,-74.102,-83.275,167.825,41.101,157.645
C08502=1032.347,-73.852,-83.287,167.828,41.100,157.645
C08503=1032.354,-73.602,-83.299,167.831,41.099,157.645
C08504=1032.359,-73.353,-83.310,167.833,41.098,157.645
C08505=1032.366,-73.103,-83.321,167.836,41.096,157.645
C08506=1032.371,-72.853,-83.332,167.839,41.095,157.645
C08507=1032.377,-72.604,-83.343,167.841,41.094,157.645
C08508=1032.383,-72.354,-83.355,167.844,41.093,157.645
C08509=1032.389,-72.104,-83.366,167.847,41.092,157.645
C08510=1032.395,-71.855,-83.378,167.850,41.091,157.645
C08511=1032.401,-71.605,-83.389,167.852,41.090,157.645
C08512=1032.408,-71.355,-83.400,167.855,41.089,157.645
C08513=1032.413,-71.106,-83.412,167.857,41.088,157.645
C08514=1032.419,-70.856,-83.424,167.860,41.087,157.645
C08515=1032.425,-70.606,-83.435,167.863,41.086,157.645
C08516=1032.432,-70.357,-83.446,167.866,41.085,157.645
C08517=1032.437,-70.107,-83.457,167.869,41.084,157.645
C08518=1032.444,-69.857,-83.469,167.871,41.082,157.645
C08519=1032.449,-69.608,-83.481,167.873,41.081,157.645
C08520=1032.455,-69.358,-83.492,167.876,41.080,157.645
C08521=1032.461,-69.109,-83.504,167.879,41.079,157.645
C08522=1032.468,-68.858,-83.515,167.882,41.078,157.644
C08523=1032.474,-68.576,-83.528,167.885,41.077,157.644
C08524=1032.481,-68.293,-83.541,167.888,41.076,157.644
C08525=1032.488,-68.010,-83.554,167.890,41.074,157.644
C08526=1032.495,-67.728,-83.567,167.894,41.073,157.644
C08527=1032.501,-67.479,-83.578,167.896,41.072,157.644
C08528=1032.507,-67.229,-83.590,167.899,41.071,157.644
C08529=1032.512,-66.980,-83.602,167.902,41.070,157.644
C08530=1032.519,-66.729,-83.613,167.905,41.069,157.644
C08531=1032.525,-66.480,-83.625,167.908,41.068,157.644
C08532=1032.531,-66.230,-83.636,167.911,41.067,157.644
///RCONF 1,0,0,0,0,0,0,0,0,0,0,0,0,0,0,0,0,0,0,0,0,0,0,0
C08533=1032.538,-65.981,-83.648,167.913,41.066,157.644
C08534=1032.543,-65.731,-83.659,167.915,41.065,157.644
C08535=1032.549,-65.481,-83.671,167.918,41.064,157.644
C08536=1032.556,-65.231,-83.683,167.921,41.063,157.644
C08537=1032.562,-64.982,-83.694,167.924,41.062,157.644
C08538=1032.567,-64.732,-83.706,167.926,41.061,157.644
C08539=1032.573,-64.483,-83.718,167.929,41.060,157.644
C08540=1032.580,-64.233,-83.730,167.932,41.059,157.644
C08541=1032.586,-63.983,-83.741,167.934,41.058,157.644
C08542=1032.592,-63.734,-83.753,167.937,41.057,157.644
C08543=1032.598,-63.484,-83.764,167.939,41.056,157.644
C08544=1032.605,-63.234,-83.776,167.942,41.055,157.644
C08545=1032.611,-62.985,-83.788,167.945,41.054,157.643
C08546=1032.617,-62.735,-83.799,167.948,41.053,157.643
C08547=1032.623,-62.485,-83.812,167.951,41.052,157.643
C08548=1032.629,-62.236,-83.822,167.954,41.051,157.643
C08549=1032.635,-61.986,-83.834,167.955,41.049,157.643
C08550=1032.642,-61.737,-83.846,167.958,41.048,157.643
C08551=1032.647,-61.487,-83.858,167.961,41.047,157.643
C08552=1032.654,-61.237,-83.870,167.964,41.046,157.643
C08553=1032.660,-60.988,-83.882,167.967,41.045,157.643
C08554=1032.665,-60.738,-83.893,167.969,41.044,157.643
C08555=1032.672,-60.488,-83.905,167.972,41.043,157.643
C08556=1032.679,-60.239,-83.917,167.975,41.042,157.643
C08557=1032.685,-59.989,-83.929,167.977,41.041,157.643
C08558=1032.690,-59.739,-83.941,167.980,41.040,157.643
C08559=1032.697,-59.490,-83.953,167.982,41.039,157.643
C08560=1032.704,-59.240,-83.965,167.985,41.038,157.643
C08561=1032.710,-58.991,-83.977,167.988,41.037,157.643
C08562=1032.715,-58.741,-83.988,167.991,41.036,157.643
C08563=1032.722,-58.491,-84.000,167.994,41.035,157.643
C08564=1032.728,-58.242,-84.012,167.995,41.034,157.643
C08565=1032.735,-57.992,-84.024,167.998,41.033,157.643
C08566=1032.740,-57.742,-84.035,168.001,41.032,157.643
C08567=1032.747,-57.493,-84.047,168.004,41.031,157.642
C08568=1032.753,-57.243,-84.059,168.006,41.030,157.642
C08569=1032.759,-56.993,-84.072,168.009,41.029,157.642
C08570=1032.766,-56.744,-84.084,168.012,41.028,157.642
C08571=1032.772,-56.494,-84.095,168.015,41.027,157.642
C08572=1032.778,-56.245,-84.107,168.018,41.026,157.642
C08573=1032.784,-55.995,-84.119,168.019,41.025,157.642
C08574=1032.791,-55.745,-84.131,168.022,41.023,157.642
C08575=1032.798,-55.496,-84.143,168.025,41.022,157.642
C08576=1032.803,-55.246,-84.155,168.028,41.021,157.642
C08577=1032.810,-54.997,-84.167,168.031,41.020,157.642
C08578=1032.816,-54.747,-84.178,168.033,41.019,157.642
C08579=1032.822,-54.497,-84.191,168.036,41.018,157.642
C08580=1032.828,-54.247,-84.203,168.038,41.017,157.642
C08581=1032.835,-53.998,-84.215,168.041,41.016,157.642
C08582=1032.842,-53.748,-84.227,168.044,41.015,157.642
C08583=1032.847,-53.499,-84.239,168.046,41.014,157.642
C08584=1032.854,-53.249,-84.251,168.049,41.013,157.642
C08585=1032.860,-53.000,-84.263,168.052,41.012,157.642
C08586=1032.866,-52.750,-84.276,168.055,41.010,157.642
C08587=1032.874,-52.468,-84.289,168.057,41.009,157.641
C08588=1032.881,-52.187,-84.303,168.060,41.008,157.641
C08589=1032.888,-51.905,-84.316,168.063,41.007,157.641
C08590=1032.895,-51.624,-84.329,168.066,41.006,157.641
C08591=1032.901,-51.374,-84.342,168.069,41.005,157.641
C08592=1032.908,-51.125,-84.354,168.072,41.004,157.641
C08593=1032.915,-50.876,-84.366,168.075,41.003,157.641
C08594=1032.920,-50.626,-84.379,168.076,41.002,157.641
C08595=1032.927,-50.376,-84.391,168.079,41.001,157.641
C08596=1032.933,-50.127,-84.403,168.082,41.000,157.641
C08597=1032.939,-49.877,-84.416,168.084,41.000,157.641
C08598=1032.946,-49.627,-84.428,168.087,40.999,157.641
C08599=1032.951,-49.377,-84.441,168.090,40.998,157.641
C08600=1032.957,-49.127,-84.453,168.092,40.997,157.641
C08601=1032.963,-48.879,-84.465,168.095,40.996,157.641
C08602=1032.970,-48.629,-84.478,168.098,40.995,157.641
C08603=1032.976,-48.379,-84.490,168.101,40.994,157.641
C08604=1032.981,-48.129,-84.503,168.103,40.993,157.641
C08605=1032.988,-47.880,-84.515,168.105,40.992,157.641
C08606=1032.994,-47.630,-84.528,168.108,40.991,157.641
C08607=1033.000,-47.381,-84.541,168.110,40.990,157.641
C08608=1033.007,-47.131,-84.553,168.113,40.989,157.641
C08609=1033.013,-46.881,-84.565,168.116,40.989,157.641
C08610=1033.019,-46.631,-84.578,168.118,40.988,157.641
C08611=1033.026,-46.382,-84.591,168.121,40.987,157.641
C08612=1033.032,-46.133,-84.603,168.124,40.986,157.641
C08613=1033.037,-45.883,-84.616,168.126,40.985,157.641
C08614=1033.044,-45.633,-84.628,168.129,40.984,157.641
C08615=1033.050,-45.384,-84.641,168.132,40.984,157.641
C08616=1033.056,-45.134,-84.653,168.133,40.983,157.641
C08617=1033.062,-44.884,-84.666,168.136,40.982,157.641
C08618=1033.069,-44.635,-84.679,168.139,40.981,157.641
C08619=1033.075,-44.385,-84.691,168.142,40.980,157.641
C08620=1033.081,-44.135,-84.704,168.144,40.979,157.641
C08621=1033.088,-43.886,-84.716,168.147,40.978,157.641
C08622=1033.094,-43.637,-84.729,168.150,40.978,157.641
C08623=1033.100,-43.387,-84.742,168.152,40.977,157.641
C08624=1033.106,-43.137,-84.755,168.155,40.976,157.641
C08625=1033.113,-42.888,-84.767,168.158,40.975,157.640
C08626=1033.118,-42.638,-84.779,168.159,40.974,157.640
C08627=1033.125,-42.389,-84.793,168.162,40.973,157.640
C08628=1033.131,-42.139,-84.805,168.165,40.973,157.640
C08629=1033.137,-41.890,-84.818,168.167,40.972,157.640
C08630=1033.143,-41.640,-84.830,168.170,40.971,157.640
C08631=1033.149,-41.390,-84.843,168.173,40.970,157.640
C08632=1033.156,-41.141,-84.856,168.175,40.969,157.640
C08633=1033.163,-40.891,-84.869,168.178,40.968,157.640
C08634=1033.169,-40.641,-84.882,168.181,40.967,157.640
C08635=1033.175,-40.391,-84.894,168.183,40.967,157.640
C08636=1033.182,-40.142,-84.907,168.186,40.966,157.640
C08637=1033.188,-39.893,-84.920,168.188,40.965,157.640
C08638=1033.194,-39.643,-84.932,168.190,40.964,157.640
C08639=1033.200,-39.393,-84.945,168.193,40.963,157.640
C08640=1033.207,-39.144,-84.957,168.196,40.962,157.640
C08641=1033.213,-38.895,-84.971,168.198,40.961,157.640
C08642=1033.220,-38.645,-84.984,168.201,40.960,157.640
C08643=1033.225,-38.395,-84.997,168.204,40.959,157.640
C08644=1033.232,-38.145,-85.010,168.206,40.959,157.640
C08645=1033.238,-37.896,-85.023,168.209,40.958,157.640
C08646=1033.244,-37.646,-85.036,168.211,40.957,157.640
C08647=1033.250,-37.396,-85.048,168.214,40.956,157.640
C08648=1033.256,-37.147,-85.062,168.216,40.955,157.640
C08649=1033.262,-36.898,-85.075,168.218,40.955,157.640
C08650=1033.268,-36.648,-85.088,168.221,40.954,157.640
C08651=1033.276,-36.367,-85.103,168.224,40.953,157.640
C08652=1033.282,-36.086,-85.117,168.227,40.952,157.640
C08653=1033.289,-35.805,-85.133,168.230,40.952,157.640
C08654=1033.296,-35.525,-85.147,168.233,40.951,157.640
C08655=1033.303,-35.275,-85.160,168.235,40.950,157.640
C08656=1033.309,-35.025,-85.173,168.238,40.949,157.640
C08657=1033.315,-34.776,-85.186,168.240,40.949,157.640
C08658=1033.321,-34.526,-85.199,168.243,40.948,157.640
C08659=1033.328,-34.277,-85.213,168.246,40.947,157.640
C08660=1033.333,-34.027,-85.225,168.248,40.946,157.640
C08661=1033.340,-33.777,-85.239,168.250,40.945,157.640
C08662=1033.346,-33.528,-85.252,168.252,40.944,157.640
C08663=1033.352,-33.278,-85.265,168.255,40.943,157.640
C08664=1033.359,-33.029,-85.278,168.258,40.943,157.640
C08665=1033.365,-32.779,-85.292,168.260,40.942,157.640
C08666=1033.372,-32.530,-85.305,168.263,40.941,157.640
C08667=1033.378,-32.280,-85.317,168.265,40.941,157.640
C08668=1033.384,-32.030,-85.331,168.268,40.940,157.640
C08669=1033.390,-31.781,-85.344,168.271,40.939,157.640
C08670=1033.397,-31.531,-85.358,168.273,40.938,157.640
C08671=1033.403,-31.282,-85.371,168.276,40.938,157.640
C08672=1033.409,-31.032,-85.383,168.278,40.937,157.640
C08673=1033.415,-30.783,-85.397,168.280,40.936,157.640
C08674=1033.421,-30.532,-85.411,168.284,40.935,157.640
C08675=1033.427,-30.283,-85.424,168.285,40.935,157.640
C08676=1033.434,-30.034,-85.437,168.288,40.934,157.640
C08677=1033.440,-29.784,-85.451,168.290,40.933,157.640
C08678=1033.446,-29.534,-85.464,168.293,40.932,157.640
C08679=1033.453,-29.285,-85.477,168.295,40.931,157.640
C08680=1033.459,-29.036,-85.490,168.298,40.930,157.640
C08681=1033.466,-28.786,-85.504,168.301,40.929,157.640
C08682=1033.472,-28.536,-85.517,168.303,40.929,157.640
C08683=1033.478,-28.287,-85.530,168.306,40.928,157.640
C08684=1033.485,-28.037,-85.544,168.308,40.927,157.640
C08685=1033.491,-27.788,-85.557,168.311,40.927,157.640
C08686=1033.497,-27.539,-85.570,168.314,40.926,157.640
C08687=1033.504,-27.289,-85.584,168.315,40.925,157.640
C08688=1033.510,-27.039,-85.597,168.318,40.924,157.640
C08689=1033.516,-26.790,-85.611,168.320,40.924,157.640
C08690=1033.523,-26.540,-85.625,168.323,40.923,157.640
C08691=1033.529,-26.291,-85.638,168.325,40.923,157.640
C08692=1033.535,-26.041,-85.651,168.328,40.922,157.640
C08693=1033.541,-25.791,-85.666,168.330,40.921,157.640
C08694=1033.547,-25.542,-85.679,168.333,40.920,157.640
C08695=1033.553,-25.293,-85.692,168.335,40.920,157.640
C08696=1033.560,-25.042,-85.706,168.338,40.919,157.640
C08697=1033.566,-24.793,-85.720,168.340,40.918,157.640
C08698=1033.572,-24.544,-85.733,168.343,40.918,157.640
C08699=1033.578,-24.293,-85.747,168.346,40.917,157.640
C08700=1033.584,-24.044,-85.760,168.348,40.916,157.640
C08701=1033.591,-23.795,-85.774,168.351,40.916,157.640
C08702=1033.597,-23.545,-85.788,168.353,40.915,157.640
C08703=1033.603,-23.295,-85.801,168.356,40.914,157.640
C08704=1033.610,-23.046,-85.816,168.357,40.914,157.640
C08705=1033.615,-22.796,-85.829,168.360,40.913,157.640
C08706=1033.622,-22.547,-85.843,168.362,40.912,157.640
C08707=1033.628,-22.297,-85.856,168.365,40.911,157.640
C08708=1033.635,-22.048,-85.870,168.367,40.911,157.640
C08709=1033.641,-21.798,-85.884,168.370,40.910,157.640
C08710=1033.647,-21.549,-85.898,168.372,40.910,157.640
C08711=1033.653,-21.300,-85.911,168.375,40.909,157.640
C08712=1033.660,-21.049,-85.925,168.377,40.908,157.640
C08713=1033.666,-20.800,-85.939,168.380,40.908,157.640
C08714=1033.673,-20.550,-85.952,168.382,40.907,157.640
C08715=1033.679,-20.269,-85.968,168.385,40.906,157.640
C08716=1033.687,-19.987,-85.983,168.388,40.905,157.640
C08717=1033.694,-19.706,-85.999,168.391,40.904,157.640
C08718=1033.701,-19.424,-86.015,168.394,40.903,157.640
C08719=1033.707,-19.174,-86.029,168.396,40.903,157.640
C08720=1033.713,-18.925,-86.042,168.398,40.902,157.640
C08721=1033.720,-18.675,-86.056,168.400,40.902,157.640
C08722=1033.725,-18.426,-86.071,168.403,40.901,157.640
C08723=1033.732,-18.176,-86.084,168.405,40.900,157.640
C08724=1033.738,-17.927,-86.097,168.408,40.900,157.640
C08725=1033.745,-17.677,-86.112,168.410,40.899,157.640
C08726=1033.751,-17.428,-86.126,168.413,40.899,157.640
C08727=1033.758,-17.178,-86.139,168.415,40.898,157.640
C08728=1033.763,-16.928,-86.153,168.418,40.897,157.640
C08729=1033.770,-16.679,-86.168,168.420,40.896,157.640
C08730=1033.777,-16.430,-86.181,168.423,40.895,157.640
C08731=1033.783,-16.179,-86.195,168.425,40.895,157.640
C08732=1033.789,-15.931,-86.209,168.428,40.894,157.640
C08733=1033.795,-15.681,-86.223,168.430,40.893,157.640
C08734=1033.802,-15.431,-86.238,168.433,40.893,157.640
C08735=1033.808,-15.182,-86.251,168.435,40.892,157.640
C08736=1033.815,-14.932,-86.265,168.438,40.892,157.640
C08737=1033.821,-14.683,-86.280,168.439,40.891,157.640
C08738=1033.827,-14.433,-86.293,168.442,40.891,157.640
C08739=1033.833,-14.184,-86.308,168.444,40.890,157.640
C08740=1033.839,-13.933,-86.322,168.446,40.889,157.640
C08741=1033.846,-13.685,-86.336,168.449,40.888,157.640
C08742=1033.852,-13.435,-86.350,168.451,40.888,157.640
C08743=1033.858,-13.186,-86.364,168.454,40.887,157.640
C08744=1033.864,-12.936,-86.379,168.456,40.887,157.640
C08745=1033.870,-12.687,-86.393,168.459,40.886,157.640
C08746=1033.877,-12.437,-86.407,168.461,40.886,157.640
C08747=1033.883,-12.188,-86.421,168.464,40.885,157.640
C08748=1033.890,-11.938,-86.435,168.466,40.885,157.640
C08749=1033.896,-11.688,-86.450,168.468,40.884,157.640
C08750=1033.902,-11.439,-86.464,168.471,40.883,157.640
C08751=1033.909,-11.189,-86.478,168.473,40.883,157.640
C08752=1033.914,-10.940,-86.493,168.476,40.882,157.640
C08753=1033.920,-10.690,-86.507,168.478,40.882,157.640
C08754=1033.927,-10.441,-86.521,168.481,40.881,157.640
C08755=1033.933,-10.191,-86.535,168.483,40.881,157.640
C08756=1033.940,-9.942,-86.550,168.485,40.880,157.640
C08757=1033.946,-9.693,-86.564,168.488,40.879,157.640
C08758=1033.952,-9.442,-86.578,168.490,40.879,157.640
C08759=1033.959,-9.193,-86.593,168.493,40.878,157.640
C08760=1033.965,-8.944,-86.607,168.494,40.877,157.640
C08761=1033.971,-8.694,-86.621,168.497,40.877,157.640
C08762=1033.978,-8.445,-86.635,168.499,40.876,157.640
C08763=1033.984,-8.195,-86.650,168.502,40.876,157.640
C08764=1033.990,-7.945,-86.665,168.504,40.875,157.640
C08765=1033.997,-7.697,-86.679,168.506,40.875,157.640
C08766=1034.003,-7.446,-86.693,168.509,40.874,157.640
C08767=1034.010,-7.197,-86.707,168.511,40.873,157.640
C08768=1034.016,-6.948,-86.722,168.514,40.872,157.640
C08769=1034.022,-6.698,-86.737,168.516,40.872,157.640
C08770=1034.029,-6.448,-86.750,168.519,40.871,157.640
C08771=1034.034,-6.200,-86.765,168.521,40.870,157.640
C08772=1034.041,-5.950,-86.780,168.523,40.870,157.640
C08773=1034.048,-5.700,-86.794,168.526,40.869,157.640
C08774=1034.054,-5.450,-86.808,168.528,40.869,157.640
C08775=1034.060,-5.201,-86.823,168.531,40.868,157.640
C08776=1034.067,-4.952,-86.837,168.533,40.868,157.640
C08777=1034.073,-4.702,-86.852,168.536,40.867,157.640
C08778=1034.079,-4.453,-86.866,168.538,40.866,157.640
C08779=1034.086,-4.169,-86.883,168.541,40.865,157.640
C08780=1034.094,-3.887,-86.899,168.543,40.865,157.640
C08781=1034.102,-3.603,-86.916,168.545,40.864,157.640
C08782=1034.108,-3.319,-86.933,168.548,40.864,157.640
C08783=1034.114,-3.070,-86.947,168.550,40.863,157.640
C08784=1034.120,-2.820,-86.962,168.553,40.863,157.640
C08785=1034.127,-2.570,-86.977,168.555,40.862,157.640
C08786=1034.132,-2.322,-86.992,168.557,40.862,157.640
C08787=1034.139,-2.072,-87.007,168.560,40.861,157.640
C08788=1034.145,-1.822,-87.022,168.562,40.861,157.640
C08789=1034.151,-1.573,-87.036,168.564,40.860,157.640
C08790=1034.157,-1.324,-87.051,168.567,40.860,157.640
C08791=1034.164,-1.074,-87.066,168.569,40.860,157.640
C08792=1034.170,-0.824,-87.080,168.571,40.859,157.640
C08793=1034.176,-0.575,-87.095,168.574,40.858,157.640
C08794=1034.182,-0.325,-87.110,168.576,40.858,157.641
C08795=1034.188,-0.075,-87.125,168.578,40.857,157.640
C08796=1034.195,0.174,-87.140,168.581,40.857,157.641
C08797=1034.200,0.423,-87.154,168.583,40.857,157.641
C08798=1034.207,0.673,-87.169,168.586,40.856,157.641
C08799=1034.213,0.923,-87.184,168.588,40.855,157.641
C08800=1034.220,1.172,-87.199,168.590,40.855,157.641
C08801=1034.226,1.421,-87.214,168.593,40.854,157.641
C08802=1034.232,1.670,-87.229,168.595,40.854,157.641
C08803=1034.238,1.920,-87.244,168.597,40.854,157.641
C08804=1034.245,2.170,-87.259,168.600,40.853,157.641
C08805=1034.251,2.419,-87.274,168.602,40.853,157.641
C08806=1034.257,2.668,-87.289,168.604,40.852,157.641
C08807=1034.263,2.918,-87.304,168.607,40.851,157.641
C08808=1034.270,3.167,-87.319,168.609,40.851,157.641
C08809=1034.276,3.417,-87.334,168.611,40.850,157.641
C08810=1034.283,3.667,-87.349,168.614,40.850,157.641
C08811=1034.288,3.916,-87.363,168.616,40.850,157.641
C08812=1034.295,4.165,-87.378,168.618,40.849,157.641
C08813=1034.301,4.415,-87.393,168.621,40.848,157.641
C08814=1034.308,4.664,-87.409,168.623,40.848,157.641
C08815=1034.314,4.914,-87.424,168.625,40.847,157.641
C08816=1034.321,5.163,-87.439,168.628,40.847,157.641
C08817=1034.326,5.412,-87.453,168.629,40.846,157.641
C08818=1034.333,5.662,-87.468,168.632,40.846,157.641
C08819=1034.339,5.912,-87.483,168.635,40.846,157.641
C08820=1034.346,6.161,-87.499,168.636,40.845,157.641
C08821=1034.352,6.410,-87.514,168.638,40.844,157.641
C08822=1034.359,6.660,-87.529,168.641,40.844,157.641
C08823=1034.365,6.910,-87.544,168.643,40.843,157.641
C08824=1034.371,7.159,-87.559,168.645,40.843,157.641
C08825=1034.377,7.408,-87.574,168.648,40.842,157.641
C08826=1034.384,7.657,-87.589,168.650,40.842,157.641
C08827=1034.390,7.907,-87.604,168.653,40.841,157.641
C08828=1034.397,8.157,-87.619,168.655,40.841,157.641
C08829=1034.403,8.406,-87.634,168.657,40.840,157.641
C08830=1034.409,8.656,-87.650,168.660,40.839,157.641
C08831=1034.415,8.905,-87.665,168.662,40.839,157.641
C08832=1034.422,9.155,-87.680,168.664,40.839,157.641
C08833=1034.428,9.404,-87.695,168.667,40.838,157.641
C08834=1034.435,9.654,-87.710,168.669,40.838,157.641
C08835=1034.441,9.903,-87.725,168.671,40.837,157.641
C08836=1034.448,10.153,-87.740,168.674,40.836,157.641
C08837=1034.454,10.402,-87.756,168.676,40.836,157.641
C08838=1034.461,10.652,-87.771,168.678,40.835,157.641
C08839=1034.466,10.901,-87.785,168.681,40.835,157.641
C08840=1034.473,11.150,-87.801,168.683,40.834,157.641
C08841=1034.479,11.399,-87.816,168.685,40.834,157.641
C08842=1034.486,11.649,-87.831,168.688,40.833,157.641
C08843=1034.493,11.934,-87.849,168.690,40.833,157.642
C08844=1034.501,12.219,-87.866,168.693,40.832,157.641
C08845=1034.508,12.505,-87.884,168.696,40.831,157.642
C08846=1034.516,12.790,-87.901,168.698,40.830,157.641
C08847=1034.522,13.039,-87.917,168.701,40.830,157.642
C08848=1034.529,13.289,-87.932,168.702,40.829,157.642
C08849=1034.535,13.539,-87.947,168.704,40.829,157.642
C08850=1034.541,13.788,-87.963,168.707,40.829,157.642
C08851=1034.547,14.038,-87.978,168.709,40.828,157.642
C08852=1034.554,14.287,-87.993,168.711,40.828,157.642
C08853=1034.561,14.536,-88.008,168.713,40.827,157.642
C08854=1034.566,14.786,-88.025,168.716,40.826,157.642
C08855=1034.573,15.035,-88.040,168.718,40.826,157.642
C08856=1034.580,15.285,-88.055,168.720,40.826,157.642
C08857=1034.585,15.534,-88.071,168.723,40.826,157.642
C08858=1034.592,15.784,-88.086,168.725,40.825,157.642
C08859=1034.598,16.033,-88.101,168.727,40.825,157.642
C08860=1034.604,16.283,-88.118,168.729,40.824,157.642
C08861=1034.611,16.532,-88.133,168.732,40.823,157.642
C08862=1034.617,16.781,-88.148,168.734,40.823,157.642
C08863=1034.623,17.031,-88.165,168.736,40.823,157.642
C08864=1034.630,17.280,-88.180,168.738,40.822,157.642
C08865=1034.636,17.529,-88.195,168.741,40.822,157.642
C08866=1034.642,17.779,-88.211,168.743,40.821,157.642
C08867=1034.649,18.028,-88.226,168.745,40.821,157.642
C08868=1034.654,18.278,-88.242,168.748,40.820,157.642
C08869=1034.661,18.527,-88.258,168.750,40.820,157.642
C08870=1034.668,18.776,-88.273,168.752,40.820,157.642
C08871=1034.673,19.026,-88.289,168.754,40.819,157.642
C08872=1034.680,19.275,-88.304,168.757,40.819,157.642
C08873=1034.687,19.524,-88.320,168.759,40.818,157.642
C08874=1034.693,19.775,-88.336,168.761,40.817,157.642
C08875=1034.700,20.024,-88.352,168.763,40.817,157.642
C08876=1034.706,20.273,-88.368,168.766,40.817,157.642
C08877=1034.712,20.523,-88.383,168.768,40.817,157.642
C08878=1034.718,20.772,-88.399,168.770,40.816,157.642
C08879=1034.725,21.021,-88.415,168.772,40.816,157.642
C08880=1034.730,21.271,-88.430,168.775,40.815,157.642
C08881=1034.737,21.520,-88.446,168.777,40.815,157.643
C08882=1034.743,21.770,-88.462,168.779,40.814,157.642
C08883=1034.750,22.019,-88.478,168.781,40.814,157.643
C08884=1034.755,22.269,-88.493,168.784,40.814,157.643
C08885=1034.762,22.518,-88.509,168.786,40.813,157.643
C08886=1034.768,22.768,-88.526,168.788,40.812,157.643
C08887=1034.775,23.017,-88.541,168.790,40.812,157.643
C08888=1034.781,23.267,-88.557,168.793,40.812,157.643
C08889=1034.787,23.516,-88.573,168.795,40.811,157.643
C08890=1034.793,23.765,-88.589,168.797,40.811,157.643
C08891=1034.800,24.014,-88.605,168.799,40.811,157.643
C08892=1034.806,24.264,-88.621,168.802,40.810,157.643
C08893=1034.813,24.513,-88.637,168.804,40.809,157.643
C08894=1034.819,24.763,-88.652,168.806,40.809,157.643
C08895=1034.826,25.012,-88.668,168.808,40.809,157.643
C08896=1034.832,25.262,-88.684,168.811,40.808,157.643
C08897=1034.838,25.511,-88.700,168.813,40.808,157.643
C08898=1034.844,25.760,-88.716,168.815,40.807,157.643
C08899=1034.852,26.010,-88.732,168.817,40.807,157.643
C08900=1034.857,26.260,-88.748,168.820,40.806,157.643
C08901=1034.864,26.509,-88.763,168.822,40.806,157.643
C08902=1034.870,26.758,-88.780,168.824,40.806,157.643
C08903=1034.877,27.007,-88.795,168.825,40.805,157.643
C08904=1034.883,27.257,-88.812,168.829,40.805,157.643
C08905=1034.889,27.507,-88.828,168.831,40.804,157.643
C08906=1034.896,27.756,-88.844,168.833,40.804,157.643
C08907=1034.903,28.042,-88.863,168.835,40.803,157.643
C08908=1034.910,28.329,-88.880,168.837,40.803,157.643
C08909=1034.918,28.615,-88.899,168.841,40.803,157.643
C08910=1034.924,28.902,-88.918,168.843,40.802,157.643
C08911=1034.931,29.151,-88.934,168.844,40.802,157.643
C08912=1034.937,29.400,-88.950,168.847,40.801,157.643
C08913=1034.943,29.650,-88.967,168.849,40.801,157.644
C08914=1034.949,29.899,-88.983,168.852,40.801,157.644
C08915=1034.956,30.148,-88.999,168.854,40.801,157.644
C08916=1034.962,30.398,-89.015,168.856,40.800,157.644
C08917=1034.969,30.648,-89.032,168.858,40.799,157.644
C08918=1034.975,30.897,-89.048,168.860,40.799,157.644
C08919=1034.981,31.146,-89.064,168.862,40.799,157.644
C08920=1034.987,31.396,-89.080,168.865,40.799,157.644
C08921=1034.993,31.645,-89.096,168.867,40.798,157.644
C08922=1035.000,31.895,-89.113,168.869,40.797,157.644
C08923=1035.006,32.144,-89.128,168.871,40.797,157.644
C08924=1035.012,32.393,-89.145,168.873,40.797,157.644
C08925=1035.019,32.642,-89.162,168.875,40.797,157.644
C08926=1035.025,32.892,-89.178,168.878,40.796,157.644
C08927=1035.032,33.141,-89.194,168.880,40.796,157.644
C08928=1035.038,33.391,-89.210,168.882,40.795,157.644
C08929=1035.044,33.641,-89.227,168.884,40.795,157.644
C08930=1035.050,33.890,-89.243,168.886,40.795,157.644
C08931=1035.057,34.139,-89.259,168.889,40.794,157.644
C08932=1035.063,34.388,-89.276,168.891,40.794,157.644
C08933=1035.070,34.638,-89.292,168.893,40.793,157.644
C08934=1035.076,34.887,-89.309,168.895,40.793,157.644
C08935=1035.082,35.136,-89.325,168.897,40.792,157.644
C08936=1035.089,35.386,-89.341,168.900,40.792,157.644
C08937=1035.095,35.636,-89.357,168.902,40.792,157.644
C08938=1035.101,35.884,-89.374,168.904,40.792,157.644
C08939=1035.108,36.134,-89.391,168.906,40.791,157.644
C08940=1035.114,36.383,-89.406,168.908,40.790,157.644
C08941=1035.120,36.633,-89.423,168.911,40.790,157.645
C08942=1035.127,36.882,-89.440,168.913,40.790,157.645
C08943=1035.133,37.131,-89.456,168.915,40.789,157.645
C08944=1035.139,37.381,-89.472,168.917,40.789,157.645
C08945=1035.146,37.631,-89.489,168.919,40.789,157.645
C08946=1035.152,37.880,-89.506,168.922,40.788,157.645
C08947=1035.158,38.129,-89.522,168.924,40.788,157.645
C08948=1035.164,38.379,-89.539,168.926,40.788,157.645
C08949=1035.171,38.628,-89.556,168.928,40.788,157.645
C08950=1035.177,38.877,-89.572,168.930,40.787,157.645
C08951=1035.183,39.127,-89.589,168.932,40.786,157.645
C08952=1035.189,39.376,-89.606,168.935,40.786,157.645
C08953=1035.195,39.625,-89.622,168.937,40.786,157.645
C08954=1035.202,39.875,-89.639,168.939,40.786,157.645
C08955=1035.208,40.124,-89.656,168.941,40.785,157.645
C08956=1035.214,40.373,-89.672,168.943,40.785,157.645
C08957=1035.221,40.623,-89.689,168.945,40.784,157.645
C08958=1035.227,40.872,-89.705,168.948,40.784,157.645
C08959=1035.233,41.121,-89.722,168.950,40.784,157.645
C08960=1035.240,41.371,-89.739,168.952,40.784,157.645
C08961=1035.246,41.620,-89.755,168.954,40.783,157.645
C08962=1035.253,41.870,-89.773,168.956,40.783,157.645
C08963=1035.259,42.119,-89.789,168.958,40.783,157.645
C08964=1035.265,42.368,-89.806,168.961,40.782,157.645
C08965=1035.271,42.618,-89.822,168.963,40.782,157.645
C08966=1035.277,42.867,-89.839,168.965,40.782,157.646
C08967=1035.284,43.117,-89.856,168.967,40.781,157.646
C08968=1035.290,43.366,-89.872,168.969,40.781,157.646
C08969=1035.296,43.615,-89.889,168.971,40.781,157.646
C08970=1035.303,43.864,-89.907,168.973,40.781,157.646
C08971=1035.310,44.151,-89.926,168.976,40.780,157.646
C08972=1035.317,44.437,-89.945,168.979,40.780,157.646
C08973=1035.324,44.724,-89.965,168.982,40.780,157.646
C08974=1035.331,45.010,-89.985,168.984,40.780,157.646
C08975=1035.337,45.259,-90.002,168.986,40.779,157.646
C08976=1035.344,45.509,-90.018,168.988,40.779,157.646
C08977=1035.349,45.758,-90.036,168.991,40.779,157.646
C08978=1035.355,46.007,-90.053,168.993,40.779,157.646
C08979=1035.362,46.257,-90.069,168.995,40.778,157.646
C08980=1035.367,46.506,-90.087,168.997,40.777,157.646
C08981=1035.374,46.756,-90.104,168.999,40.777,157.646
C08982=1035.380,47.005,-90.121,169.001,40.777,157.646
C08983=1035.387,47.254,-90.138,169.003,40.777,157.646
C08984=1035.392,47.504,-90.155,169.006,40.776,157.647
C08985=1035.399,47.753,-90.172,169.008,40.776,157.647
C08986=1035.405,48.002,-90.189,169.010,40.776,157.647
C08987=1035.411,48.252,-90.206,169.012,40.776,157.647
C08988=1035.418,48.501,-90.223,169.014,40.776,157.647
C08989=1035.424,48.750,-90.240,169.016,40.775,157.647
C08990=1035.430,49.000,-90.257,169.018,40.775,157.647
C08991=1035.436,49.249,-90.274,169.020,40.775,157.647
C08992=1035.443,49.498,-90.292,169.023,40.775,157.647
C08993=1035.449,49.747,-90.309,169.025,40.774,157.647
C08994=1035.455,49.998,-90.326,169.027,40.774,157.647
C08995=1035.461,50.246,-90.343,169.029,40.774,157.647
C08996=1035.468,50.496,-90.360,169.031,40.774,157.647
C08997=1035.473,50.745,-90.378,169.033,40.773,157.647
C08998=1035.480,50.995,-90.394,169.035,40.773,157.647
C08999=1035.486,51.243,-90.411,169.037,40.772,157.647
C09000=1035.492,51.493,-90.429,169.040,40.772,157.647
C09001=1035.499,51.742,-90.446,169.042,40.772,157.647
C09002=1035.505,51.992,-90.463,169.044,40.772,157.648
C09003=1035.511,52.241,-90.480,169.046,40.771,157.648
C09004=1035.518,52.490,-90.498,169.048,40.771,157.648
C09005=1035.524,52.739,-90.515,169.050,40.771,157.648
C09006=1035.531,52.989,-90.532,169.052,40.771,157.648
C09007=1035.536,53.238,-90.550,169.055,40.770,157.648
C09008=1035.543,53.488,-90.566,169.057,40.769,157.648
C09009=1035.550,53.737,-90.584,169.059,40.769,157.648
C09010=1035.555,53.986,-90.601,169.061,40.769,157.648
C09011=1035.562,54.236,-90.619,169.063,40.769,157.648
C09012=1035.568,54.484,-90.636,169.065,40.769,157.648
C09013=1035.574,54.734,-90.654,169.067,40.768,157.648
C09014=1035.580,54.983,-90.670,169.070,40.768,157.648
C09015=1035.587,55.233,-90.687,169.072,40.768,157.648
